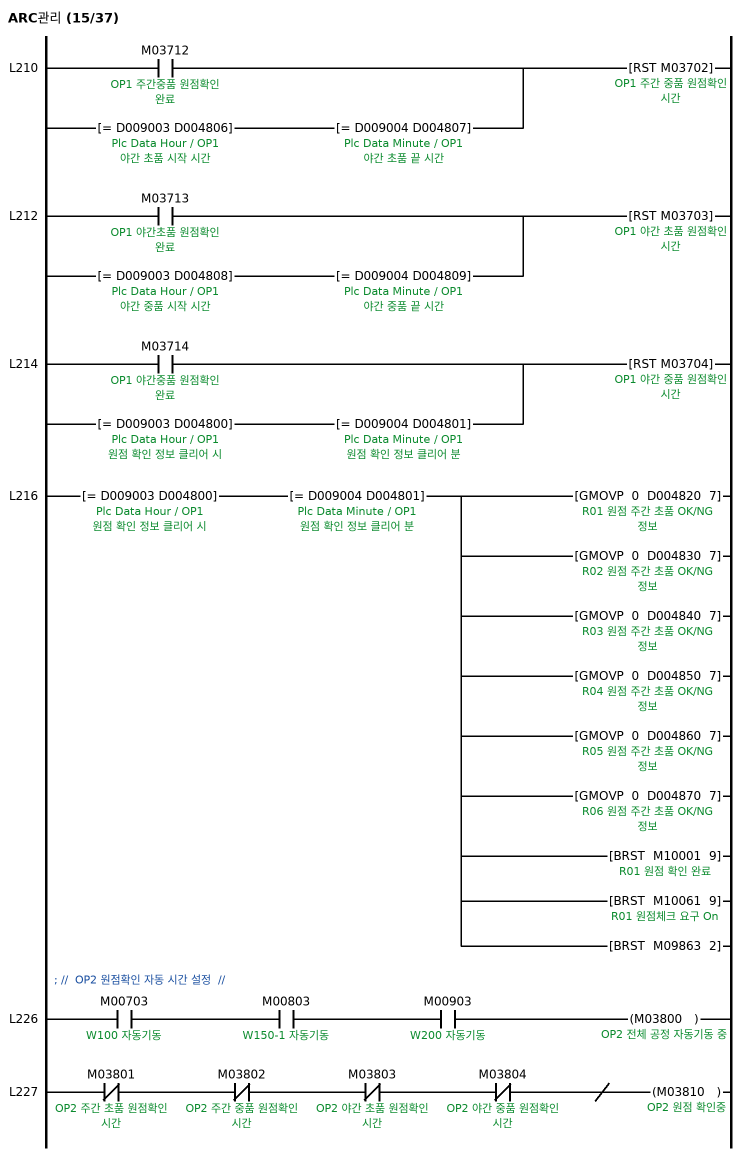
[picture p408: ARC관리 rungs L210-L227]
; L210
LOAD      M03712	// OP1 주간중품 원점확인 완료
LOAD=     D009003 D004806	// Plc Data Hour / OP1 야간 초품 시작 시간
AND=      D009004 D004807	// Plc Data Minute / OP1 야간 초품 끝 시간
OR LOAD
RST       M03702	// OP1 주간 중품 원점확인 시간
; L212
LOAD      M03713	// OP1 야간초품 원점확인 완료
LOAD=     D009003 D004808	// Plc Data Hour / OP1 야간 중품 시작 시간
AND=      D009004 D004809	// Plc Data Minute / OP1 야간 중품 끝 시간
OR LOAD
RST       M03703	// OP1 야간 초품 원점확인 시간
; L214
LOAD      M03714	// OP1 야간중품 원점확인 완료
LOAD=     D009003 D004800	// Plc Data Hour / OP1 원점 확인 정보 클리어 시
AND=      D009004 D004801	// Plc Data Minute / OP1 원점 확인 정보 클리어 분
OR LOAD
RST       M03704	// OP1 야간 중품 원점확인 시간
; L216
LOAD=     D009003 D004800	// Plc Data Hour / OP1 원점 확인 정보 클리어 시
AND=      D009004 D004801	// Plc Data Minute / OP1 원점 확인 정보 클리어 분
GMOVP     0 D004820 7	// R01 원점 주간 초품 OK/NG 정보
GMOVP     0 D004830 7	// R02 원점 주간 초품 OK/NG 정보
GMOVP     0 D004840 7	// R03 원점 주간 초품 OK/NG 정보
GMOVP     0 D004850 7	// R04 원점 주간 초품 OK/NG 정보
GMOVP     0 D004860 7	// R05 원점 주간 초품 OK/NG 정보
GMOVP     0 D004870 7	// R06 원점 주간 초품 OK/NG 정보
BRST      M10001 9	// R01 원점 확인 완료
BRST      M10061 9	// R01 원점체크 요구 On
BRST      M09863 2
//   //  OP2 원점확인 자동 시간 설정  //
; L226
LOAD      M00703	// W100 자동기동
AND       M00803	// W150-1 자동기동
AND       M00903	// W200 자동기동
OUT       M03800	// OP2 전체 공정 자동기동 중
; L227
LOAD NOT  M03801	// OP2 주간 초품 원점확인 시간
AND NOT   M03802	// OP2 주간 중품 원점확인 시간
AND NOT   M03803	// OP2 야간 초품 원점확인 시간
AND NOT   M03804	// OP2 야간 중품 원점확인 시간
NOT
OUT       M03810	// OP2 원점 확인중

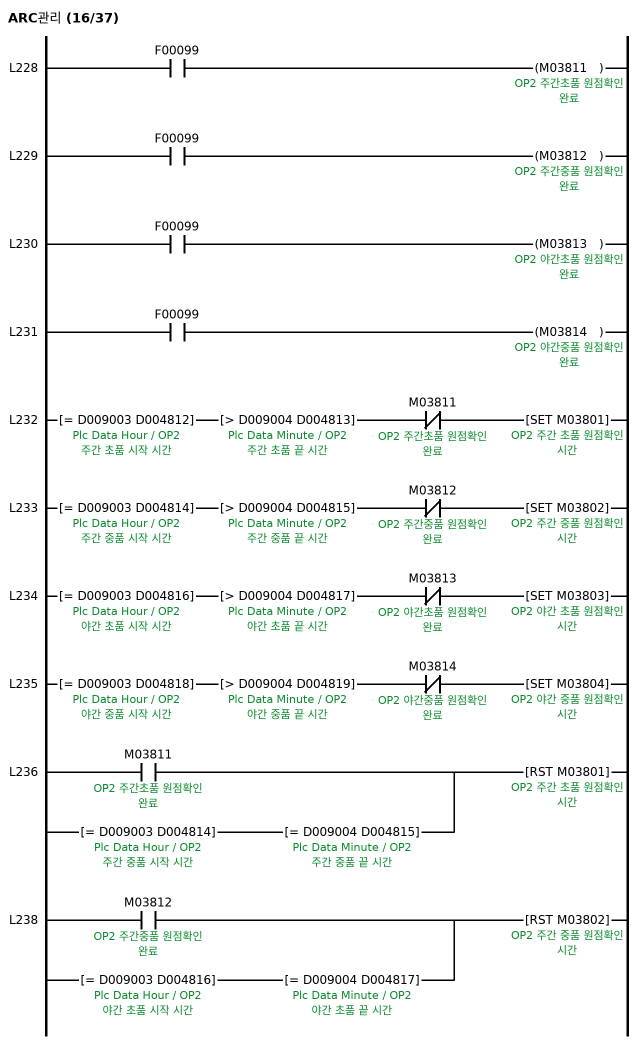
; L228
LOAD      F00099
OUT       M03811	// OP2 주간초품 원점확인 완료
; L229
LOAD      F00099
OUT       M03812	// OP2 주간중품 원점확인 완료
; L230
LOAD      F00099
OUT       M03813	// OP2 야간초품 원점확인 완료
; L231
LOAD      F00099
OUT       M03814	// OP2 야간중품 원점확인 완료
; L232
LOAD=     D009003 D004812	// Plc Data Hour / OP2 주간 초품 시작 시간
AND>      D009004 D004813	// Plc Data Minute / OP2 주간 초품 끝 시간
AND NOT   M03811	// OP2 주간초품 원점확인 완료
SET       M03801	// OP2 주간 초품 원점확인 시간
; L233
LOAD=     D009003 D004814	// Plc Data Hour / OP2 주간 중품 시작 시간
AND>      D009004 D004815	// Plc Data Minute / OP2 주간 중품 끝 시간
AND NOT   M03812	// OP2 주간중품 원점확인 완료
SET       M03802	// OP2 주간 중품 원점확인 시간
; L234
LOAD=     D009003 D004816	// Plc Data Hour / OP2 야간 초품 시작 시간
AND>      D009004 D004817	// Plc Data Minute / OP2 야간 초품 끝 시간
AND NOT   M03813	// OP2 야간초품 원점확인 완료
SET       M03803	// OP2 야간 초품 원점확인 시간
; L235
LOAD=     D009003 D004818	// Plc Data Hour / OP2 야간 중품 시작 시간
AND>      D009004 D004819	// Plc Data Minute / OP2 야간 중품 끝 시간
AND NOT   M03814	// OP2 야간중품 원점확인 완료
SET       M03804	// OP2 야간 중품 원점확인 시간
; L236
LOAD      M03811	// OP2 주간초품 원점확인 완료
LOAD=     D009003 D004814	// Plc Data Hour / OP2 주간 중품 시작 시간
AND=      D009004 D004815	// Plc Data Minute / OP2 주간 중품 끝 시간
OR LOAD
RST       M03801	// OP2 주간 초품 원점확인 시간
; L238
LOAD      M03812	// OP2 주간중품 원점확인 완료
LOAD=     D009003 D004816	// Plc Data Hour / OP2 야간 초품 시작 시간
AND=      D009004 D004817	// Plc Data Minute / OP2 야간 초품 끝 시간
OR LOAD
RST       M03802	// OP2 주간 중품 원점확인 시간

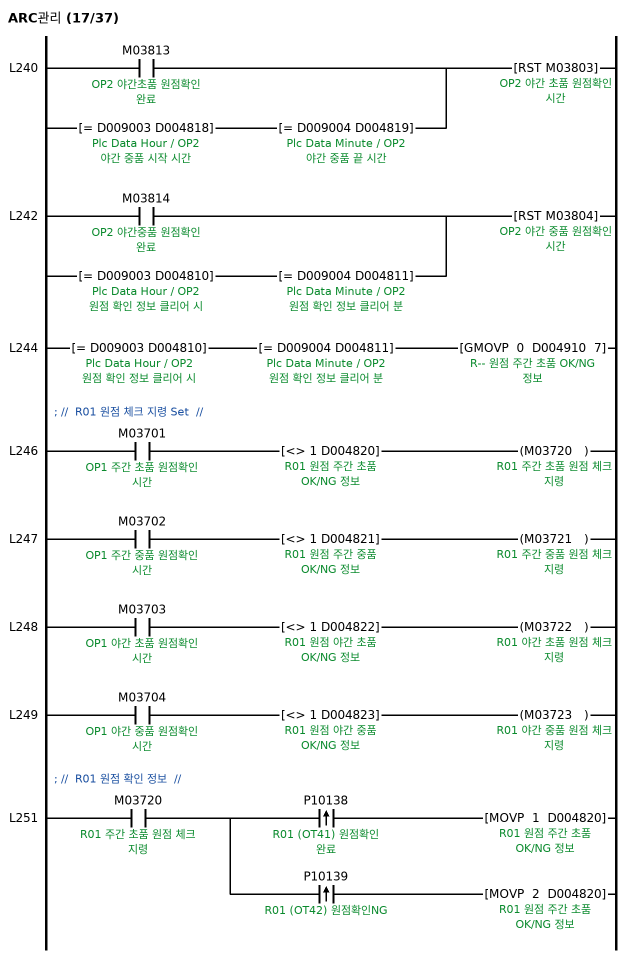
; L240
LOAD      M03813	// OP2 야간초품 원점확인 완료
LOAD=     D009003 D004818	// Plc Data Hour / OP2 야간 중품 시작 시간
AND=      D009004 D004819	// Plc Data Minute / OP2 야간 중품 끝 시간
OR LOAD
RST       M03803	// OP2 야간 초품 원점확인 시간
; L242
LOAD      M03814	// OP2 야간중품 원점확인 완료
LOAD=     D009003 D004810	// Plc Data Hour / OP2 원점 확인 정보 클리어 시
AND=      D009004 D004811	// Plc Data Minute / OP2 원점 확인 정보 클리어 분
OR LOAD
RST       M03804	// OP2 야간 중품 원점확인 시간
; L244
LOAD=     D009003 D004810	// Plc Data Hour / OP2 원점 확인 정보 클리어 시
AND=      D009004 D004811	// Plc Data Minute / OP2 원점 확인 정보 클리어 분
GMOVP     0 D004910 7	// R-- 원점 주간 초품 OK/NG 정보
//   //  R01 원점 체크 지령 Set  //
; L246
LOAD      M03701	// OP1 주간 초품 원점확인 시간
AND<>     1 D004820	// R01 원점 주간 초품 OK/NG 정보
OUT       M03720	// R01 주간 초품 원점 체크 지령
; L247
LOAD      M03702	// OP1 주간 중품 원점확인 시간
AND<>     1 D004821	// R01 원점 주간 중품 OK/NG 정보
OUT       M03721	// R01 주간 중품 원점 체크 지령
; L248
LOAD      M03703	// OP1 야간 초품 원점확인 시간
AND<>     1 D004822	// R01 원점 야간 초품 OK/NG 정보
OUT       M03722	// R01 야간 초품 원점 체크 지령
; L249
LOAD      M03704	// OP1 야간 중품 원점확인 시간
AND<>     1 D004823	// R01 원점 야간 중품 OK/NG 정보
OUT       M03723	// R01 야간 중품 원점 체크 지령
//   //  R01 원점 확인 정보  //
; L251
LOAD      M03720	// R01 주간 초품 원점 체크 지령
MPUSH
ANDP      P10138	// R01 (OT41) 원점확인 완료
MOVP      1 D004820	// R01 원점 주간 초품 OK/NG 정보
MPOP
ANDP      P10139	// R01 (OT42) 원점확인NG
MOVP      2 D004820	// R01 원점 주간 초품 OK/NG 정보

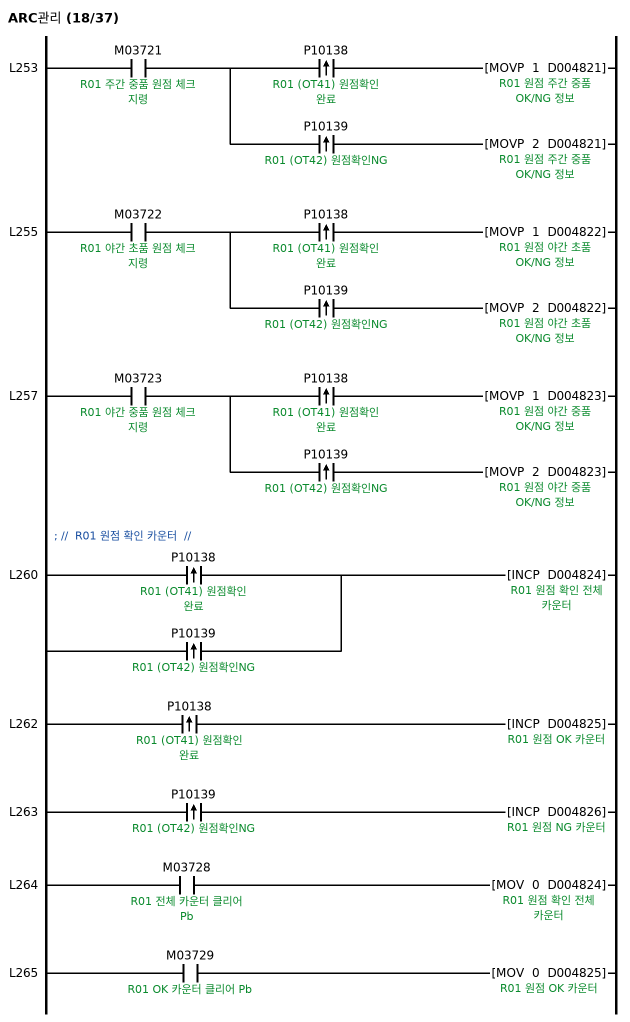
; L253
LOAD      M03721	// R01 주간 중품 원점 체크 지령
MPUSH
ANDP      P10138	// R01 (OT41) 원점확인 완료
MOVP      1 D004821	// R01 원점 주간 중품 OK/NG 정보
MPOP
ANDP      P10139	// R01 (OT42) 원점확인NG
MOVP      2 D004821	// R01 원점 주간 중품 OK/NG 정보
; L255
LOAD      M03722	// R01 야간 초품 원점 체크 지령
MPUSH
ANDP      P10138	// R01 (OT41) 원점확인 완료
MOVP      1 D004822	// R01 원점 야간 초품 OK/NG 정보
MPOP
ANDP      P10139	// R01 (OT42) 원점확인NG
MOVP      2 D004822	// R01 원점 야간 초품 OK/NG 정보
; L257
LOAD      M03723	// R01 야간 중품 원점 체크 지령
MPUSH
ANDP      P10138	// R01 (OT41) 원점확인 완료
MOVP      1 D004823	// R01 원점 야간 중품 OK/NG 정보
MPOP
ANDP      P10139	// R01 (OT42) 원점확인NG
MOVP      2 D004823	// R01 원점 야간 중품 OK/NG 정보
//   //  R01 원점 확인 카운터  //
; L260
LOADP     P10138	// R01 (OT41) 원점확인 완료
ORP       P10139	// R01 (OT42) 원점확인NG
INCP      D004824	// R01 원점 확인 전체 카운터
; L262
LOADP     P10138	// R01 (OT41) 원점확인 완료
INCP      D004825	// R01 원점 OK 카운터
; L263
LOADP     P10139	// R01 (OT42) 원점확인NG
INCP      D004826	// R01 원점 NG 카운터
; L264
LOAD      M03728	// R01 전체 카운터 클리어 Pb
MOV       0 D004824	// R01 원점 확인 전체 카운터
; L265
LOAD      M03729	// R01 OK 카운터 클리어 Pb
MOV       0 D004825	// R01 원점 OK 카운터

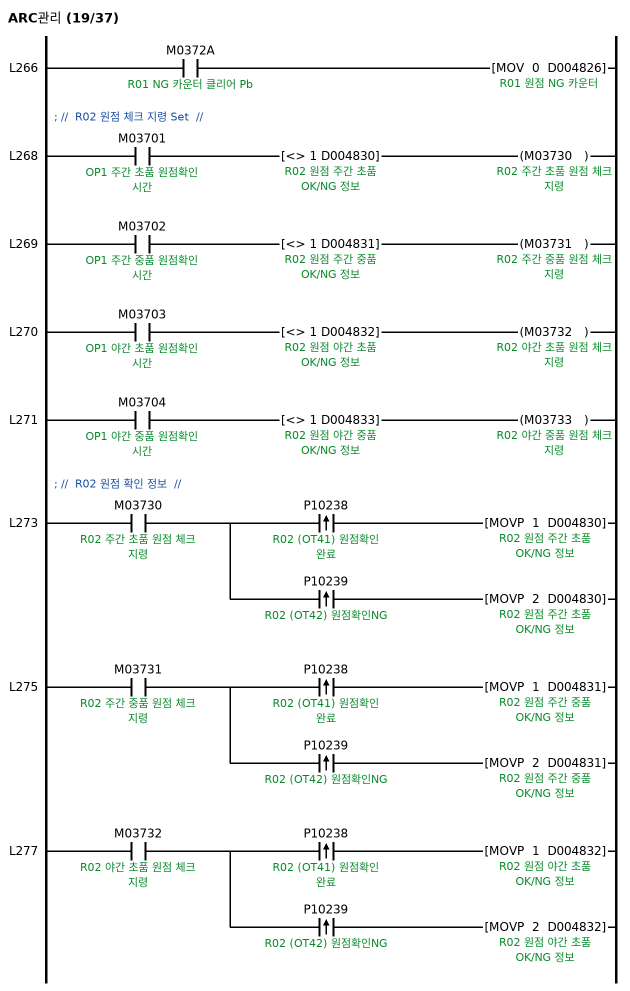
; L266
LOAD      M0372A	// R01 NG 카운터 클리어 Pb
MOV       0 D004826	// R01 원점 NG 카운터
//   //  R02 원점 체크 지령 Set  //
; L268
LOAD      M03701	// OP1 주간 초품 원점확인 시간
AND<>     1 D004830	// R02 원점 주간 초품 OK/NG 정보
OUT       M03730	// R02 주간 초품 원점 체크 지령
; L269
LOAD      M03702	// OP1 주간 중품 원점확인 시간
AND<>     1 D004831	// R02 원점 주간 중품 OK/NG 정보
OUT       M03731	// R02 주간 중품 원점 체크 지령
; L270
LOAD      M03703	// OP1 야간 초품 원점확인 시간
AND<>     1 D004832	// R02 원점 야간 초품 OK/NG 정보
OUT       M03732	// R02 야간 초품 원점 체크 지령
; L271
LOAD      M03704	// OP1 야간 중품 원점확인 시간
AND<>     1 D004833	// R02 원점 야간 중품 OK/NG 정보
OUT       M03733	// R02 야간 중품 원점 체크 지령
//   //  R02 원점 확인 정보  //
; L273
LOAD      M03730	// R02 주간 초품 원점 체크 지령
MPUSH
ANDP      P10238	// R02 (OT41) 원점확인 완료
MOVP      1 D004830	// R02 원점 주간 초품 OK/NG 정보
MPOP
ANDP      P10239	// R02 (OT42) 원점확인NG
MOVP      2 D004830	// R02 원점 주간 초품 OK/NG 정보
; L275
LOAD      M03731	// R02 주간 중품 원점 체크 지령
MPUSH
ANDP      P10238	// R02 (OT41) 원점확인 완료
MOVP      1 D004831	// R02 원점 주간 중품 OK/NG 정보
MPOP
ANDP      P10239	// R02 (OT42) 원점확인NG
MOVP      2 D004831	// R02 원점 주간 중품 OK/NG 정보
; L277
LOAD      M03732	// R02 야간 초품 원점 체크 지령
MPUSH
ANDP      P10238	// R02 (OT41) 원점확인 완료
MOVP      1 D004832	// R02 원점 야간 초품 OK/NG 정보
MPOP
ANDP      P10239	// R02 (OT42) 원점확인NG
MOVP      2 D004832	// R02 원점 야간 초품 OK/NG 정보

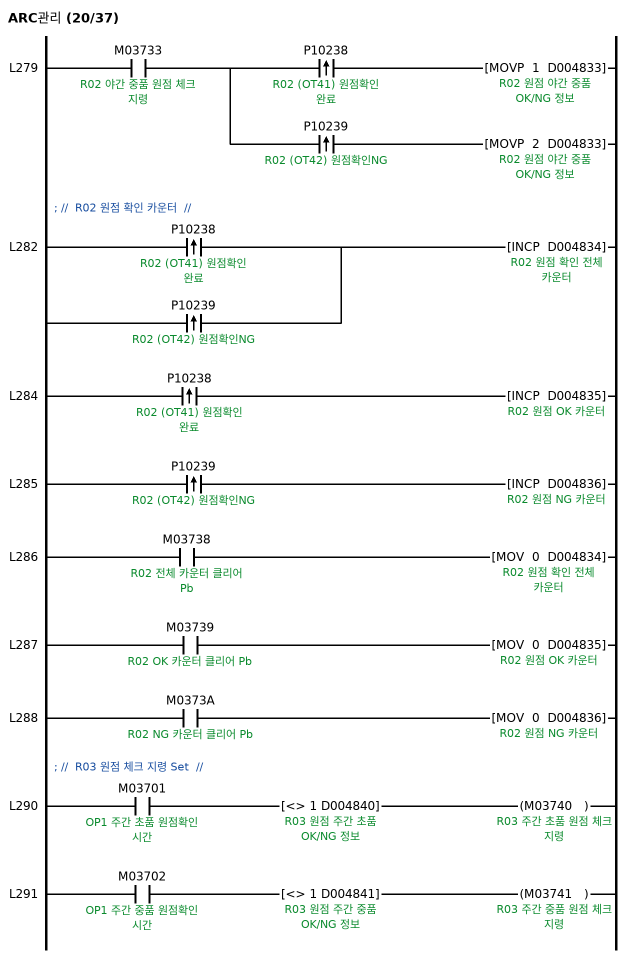
; L279
LOAD      M03733	// R02 야간 중품 원점 체크 지령
MPUSH
ANDP      P10238	// R02 (OT41) 원점확인 완료
MOVP      1 D004833	// R02 원점 야간 중품 OK/NG 정보
MPOP
ANDP      P10239	// R02 (OT42) 원점확인NG
MOVP      2 D004833	// R02 원점 야간 중품 OK/NG 정보
//   //  R02 원점 확인 카운터  //
; L282
LOADP     P10238	// R02 (OT41) 원점확인 완료
ORP       P10239	// R02 (OT42) 원점확인NG
INCP      D004834	// R02 원점 확인 전체 카운터
; L284
LOADP     P10238	// R02 (OT41) 원점확인 완료
INCP      D004835	// R02 원점 OK 카운터
; L285
LOADP     P10239	// R02 (OT42) 원점확인NG
INCP      D004836	// R02 원점 NG 카운터
; L286
LOAD      M03738	// R02 전체 카운터 클리어 Pb
MOV       0 D004834	// R02 원점 확인 전체 카운터
; L287
LOAD      M03739	// R02 OK 카운터 클리어 Pb
MOV       0 D004835	// R02 원점 OK 카운터
; L288
LOAD      M0373A	// R02 NG 카운터 클리어 Pb
MOV       0 D004836	// R02 원점 NG 카운터
//   //  R03 원점 체크 지령 Set  //
; L290
LOAD      M03701	// OP1 주간 초품 원점확인 시간
AND<>     1 D004840	// R03 원점 주간 초품 OK/NG 정보
OUT       M03740	// R03 주간 초품 원점 체크 지령
; L291
LOAD      M03702	// OP1 주간 중품 원점확인 시간
AND<>     1 D004841	// R03 원점 주간 중품 OK/NG 정보
OUT       M03741	// R03 주간 중품 원점 체크 지령

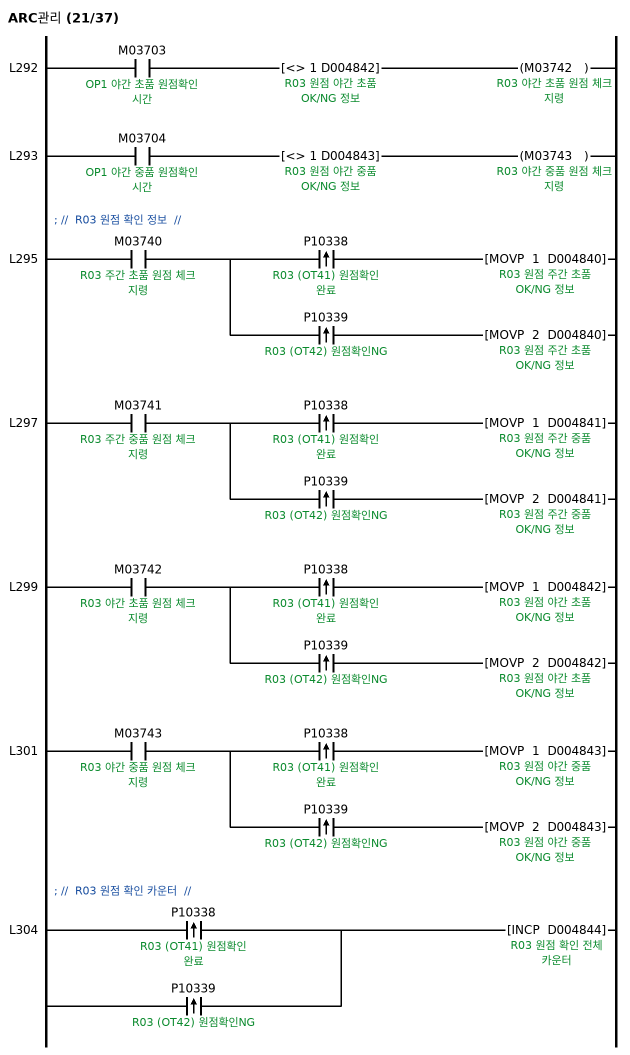
; L292
LOAD      M03703	// OP1 야간 초품 원점확인 시간
AND<>     1 D004842	// R03 원점 야간 초품 OK/NG 정보
OUT       M03742	// R03 야간 초품 원점 체크 지령
; L293
LOAD      M03704	// OP1 야간 중품 원점확인 시간
AND<>     1 D004843	// R03 원점 야간 중품 OK/NG 정보
OUT       M03743	// R03 야간 중품 원점 체크 지령
//   //  R03 원점 확인 정보  //
; L295
LOAD      M03740	// R03 주간 초품 원점 체크 지령
MPUSH
ANDP      P10338	// R03 (OT41) 원점확인 완료
MOVP      1 D004840	// R03 원점 주간 초품 OK/NG 정보
MPOP
ANDP      P10339	// R03 (OT42) 원점확인NG
MOVP      2 D004840	// R03 원점 주간 초품 OK/NG 정보
; L297
LOAD      M03741	// R03 주간 중품 원점 체크 지령
MPUSH
ANDP      P10338	// R03 (OT41) 원점확인 완료
MOVP      1 D004841	// R03 원점 주간 중품 OK/NG 정보
MPOP
ANDP      P10339	// R03 (OT42) 원점확인NG
MOVP      2 D004841	// R03 원점 주간 중품 OK/NG 정보
; L299
LOAD      M03742	// R03 야간 초품 원점 체크 지령
MPUSH
ANDP      P10338	// R03 (OT41) 원점확인 완료
MOVP      1 D004842	// R03 원점 야간 초품 OK/NG 정보
MPOP
ANDP      P10339	// R03 (OT42) 원점확인NG
MOVP      2 D004842	// R03 원점 야간 초품 OK/NG 정보
; L301
LOAD      M03743	// R03 야간 중품 원점 체크 지령
MPUSH
ANDP      P10338	// R03 (OT41) 원점확인 완료
MOVP      1 D004843	// R03 원점 야간 중품 OK/NG 정보
MPOP
ANDP      P10339	// R03 (OT42) 원점확인NG
MOVP      2 D004843	// R03 원점 야간 중품 OK/NG 정보
//   //  R03 원점 확인 카운터  //
; L304
LOADP     P10338	// R03 (OT41) 원점확인 완료
ORP       P10339	// R03 (OT42) 원점확인NG
INCP      D004844	// R03 원점 확인 전체 카운터

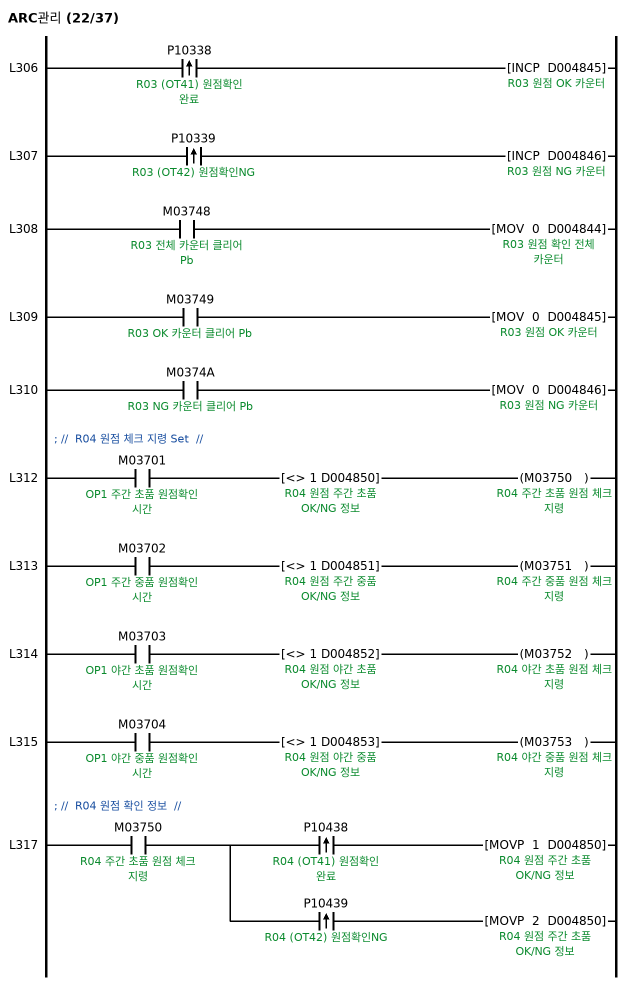
; L306
LOADP     P10338	// R03 (OT41) 원점확인 완료
INCP      D004845	// R03 원점 OK 카운터
; L307
LOADP     P10339	// R03 (OT42) 원점확인NG
INCP      D004846	// R03 원점 NG 카운터
; L308
LOAD      M03748	// R03 전체 카운터 클리어 Pb
MOV       0 D004844	// R03 원점 확인 전체 카운터
; L309
LOAD      M03749	// R03 OK 카운터 클리어 Pb
MOV       0 D004845	// R03 원점 OK 카운터
; L310
LOAD      M0374A	// R03 NG 카운터 클리어 Pb
MOV       0 D004846	// R03 원점 NG 카운터
//   //  R04 원점 체크 지령 Set  //
; L312
LOAD      M03701	// OP1 주간 초품 원점확인 시간
AND<>     1 D004850	// R04 원점 주간 초품 OK/NG 정보
OUT       M03750	// R04 주간 초품 원점 체크 지령
; L313
LOAD      M03702	// OP1 주간 중품 원점확인 시간
AND<>     1 D004851	// R04 원점 주간 중품 OK/NG 정보
OUT       M03751	// R04 주간 중품 원점 체크 지령
; L314
LOAD      M03703	// OP1 야간 초품 원점확인 시간
AND<>     1 D004852	// R04 원점 야간 초품 OK/NG 정보
OUT       M03752	// R04 야간 초품 원점 체크 지령
; L315
LOAD      M03704	// OP1 야간 중품 원점확인 시간
AND<>     1 D004853	// R04 원점 야간 중품 OK/NG 정보
OUT       M03753	// R04 야간 중품 원점 체크 지령
//   //  R04 원점 확인 정보  //
; L317
LOAD      M03750	// R04 주간 초품 원점 체크 지령
MPUSH
ANDP      P10438	// R04 (OT41) 원점확인 완료
MOVP      1 D004850	// R04 원점 주간 초품 OK/NG 정보
MPOP
ANDP      P10439	// R04 (OT42) 원점확인NG
MOVP      2 D004850	// R04 원점 주간 초품 OK/NG 정보

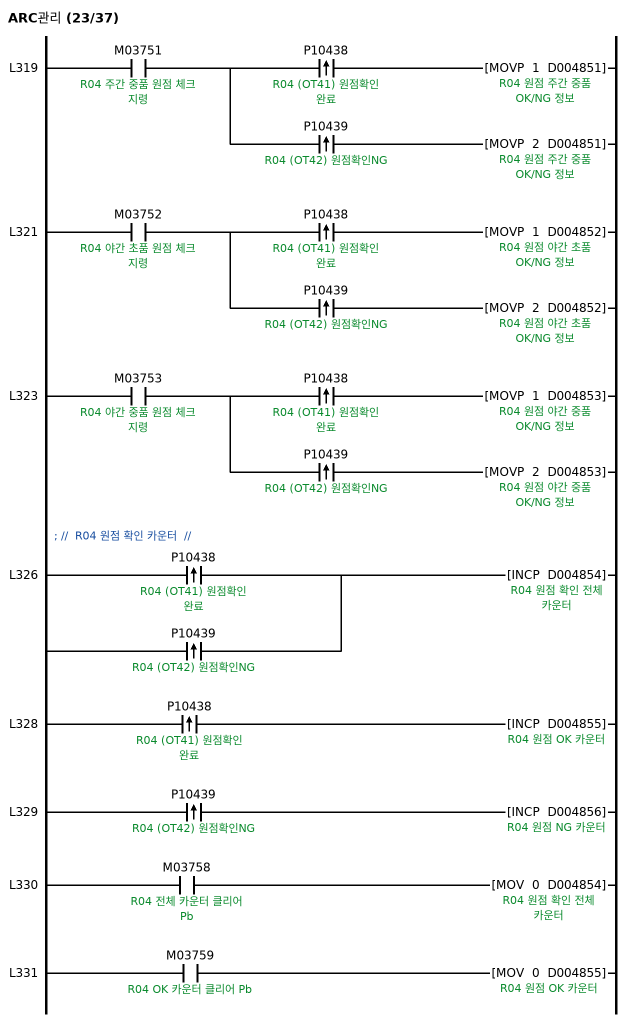
; L319
LOAD      M03751	// R04 주간 중품 원점 체크 지령
MPUSH
ANDP      P10438	// R04 (OT41) 원점확인 완료
MOVP      1 D004851	// R04 원점 주간 중품 OK/NG 정보
MPOP
ANDP      P10439	// R04 (OT42) 원점확인NG
MOVP      2 D004851	// R04 원점 주간 중품 OK/NG 정보
; L321
LOAD      M03752	// R04 야간 초품 원점 체크 지령
MPUSH
ANDP      P10438	// R04 (OT41) 원점확인 완료
MOVP      1 D004852	// R04 원점 야간 초품 OK/NG 정보
MPOP
ANDP      P10439	// R04 (OT42) 원점확인NG
MOVP      2 D004852	// R04 원점 야간 초품 OK/NG 정보
; L323
LOAD      M03753	// R04 야간 중품 원점 체크 지령
MPUSH
ANDP      P10438	// R04 (OT41) 원점확인 완료
MOVP      1 D004853	// R04 원점 야간 중품 OK/NG 정보
MPOP
ANDP      P10439	// R04 (OT42) 원점확인NG
MOVP      2 D004853	// R04 원점 야간 중품 OK/NG 정보
//   //  R04 원점 확인 카운터  //
; L326
LOADP     P10438	// R04 (OT41) 원점확인 완료
ORP       P10439	// R04 (OT42) 원점확인NG
INCP      D004854	// R04 원점 확인 전체 카운터
; L328
LOADP     P10438	// R04 (OT41) 원점확인 완료
INCP      D004855	// R04 원점 OK 카운터
; L329
LOADP     P10439	// R04 (OT42) 원점확인NG
INCP      D004856	// R04 원점 NG 카운터
; L330
LOAD      M03758	// R04 전체 카운터 클리어 Pb
MOV       0 D004854	// R04 원점 확인 전체 카운터
; L331
LOAD      M03759	// R04 OK 카운터 클리어 Pb
MOV       0 D004855	// R04 원점 OK 카운터

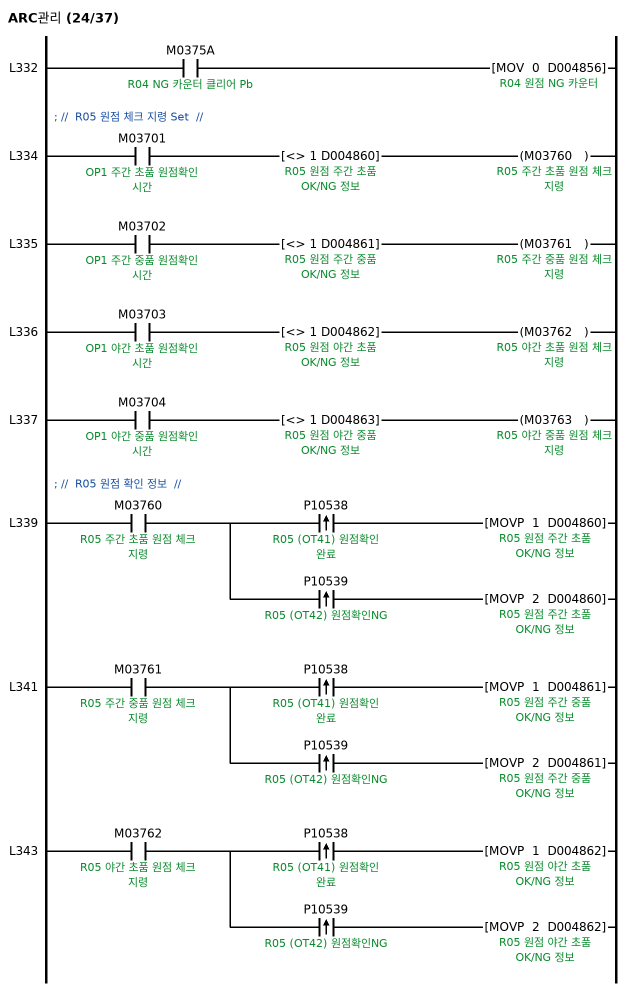
; L332
LOAD      M0375A	// R04 NG 카운터 클리어 Pb
MOV       0 D004856	// R04 원점 NG 카운터
//   //  R05 원점 체크 지령 Set  //
; L334
LOAD      M03701	// OP1 주간 초품 원점확인 시간
AND<>     1 D004860	// R05 원점 주간 초품 OK/NG 정보
OUT       M03760	// R05 주간 초품 원점 체크 지령
; L335
LOAD      M03702	// OP1 주간 중품 원점확인 시간
AND<>     1 D004861	// R05 원점 주간 중품 OK/NG 정보
OUT       M03761	// R05 주간 중품 원점 체크 지령
; L336
LOAD      M03703	// OP1 야간 초품 원점확인 시간
AND<>     1 D004862	// R05 원점 야간 초품 OK/NG 정보
OUT       M03762	// R05 야간 초품 원점 체크 지령
; L337
LOAD      M03704	// OP1 야간 중품 원점확인 시간
AND<>     1 D004863	// R05 원점 야간 중품 OK/NG 정보
OUT       M03763	// R05 야간 중품 원점 체크 지령
//   //  R05 원점 확인 정보  //
; L339
LOAD      M03760	// R05 주간 초품 원점 체크 지령
MPUSH
ANDP      P10538	// R05 (OT41) 원점확인 완료
MOVP      1 D004860	// R05 원점 주간 초품 OK/NG 정보
MPOP
ANDP      P10539	// R05 (OT42) 원점확인NG
MOVP      2 D004860	// R05 원점 주간 초품 OK/NG 정보
; L341
LOAD      M03761	// R05 주간 중품 원점 체크 지령
MPUSH
ANDP      P10538	// R05 (OT41) 원점확인 완료
MOVP      1 D004861	// R05 원점 주간 중품 OK/NG 정보
MPOP
ANDP      P10539	// R05 (OT42) 원점확인NG
MOVP      2 D004861	// R05 원점 주간 중품 OK/NG 정보
; L343
LOAD      M03762	// R05 야간 초품 원점 체크 지령
MPUSH
ANDP      P10538	// R05 (OT41) 원점확인 완료
MOVP      1 D004862	// R05 원점 야간 초품 OK/NG 정보
MPOP
ANDP      P10539	// R05 (OT42) 원점확인NG
MOVP      2 D004862	// R05 원점 야간 초품 OK/NG 정보

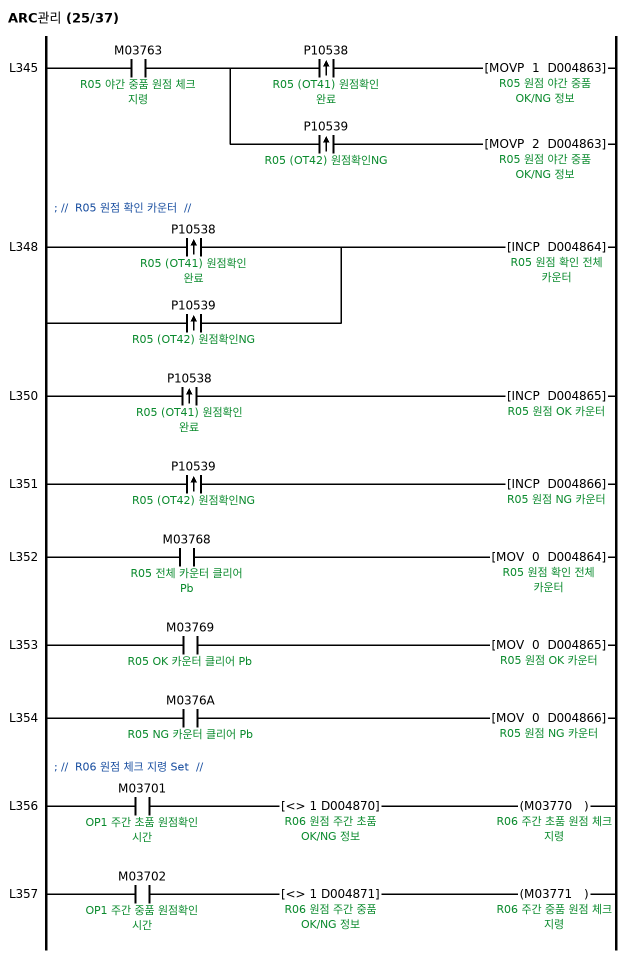
; L345
LOAD      M03763	// R05 야간 중품 원점 체크 지령
MPUSH
ANDP      P10538	// R05 (OT41) 원점확인 완료
MOVP      1 D004863	// R05 원점 야간 중품 OK/NG 정보
MPOP
ANDP      P10539	// R05 (OT42) 원점확인NG
MOVP      2 D004863	// R05 원점 야간 중품 OK/NG 정보
//   //  R05 원점 확인 카운터  //
; L348
LOADP     P10538	// R05 (OT41) 원점확인 완료
ORP       P10539	// R05 (OT42) 원점확인NG
INCP      D004864	// R05 원점 확인 전체 카운터
; L350
LOADP     P10538	// R05 (OT41) 원점확인 완료
INCP      D004865	// R05 원점 OK 카운터
; L351
LOADP     P10539	// R05 (OT42) 원점확인NG
INCP      D004866	// R05 원점 NG 카운터
; L352
LOAD      M03768	// R05 전체 카운터 클리어 Pb
MOV       0 D004864	// R05 원점 확인 전체 카운터
; L353
LOAD      M03769	// R05 OK 카운터 클리어 Pb
MOV       0 D004865	// R05 원점 OK 카운터
; L354
LOAD      M0376A	// R05 NG 카운터 클리어 Pb
MOV       0 D004866	// R05 원점 NG 카운터
//   //  R06 원점 체크 지령 Set  //
; L356
LOAD      M03701	// OP1 주간 초품 원점확인 시간
AND<>     1 D004870	// R06 원점 주간 초품 OK/NG 정보
OUT       M03770	// R06 주간 초품 원점 체크 지령
; L357
LOAD      M03702	// OP1 주간 중품 원점확인 시간
AND<>     1 D004871	// R06 원점 주간 중품 OK/NG 정보
OUT       M03771	// R06 주간 중품 원점 체크 지령

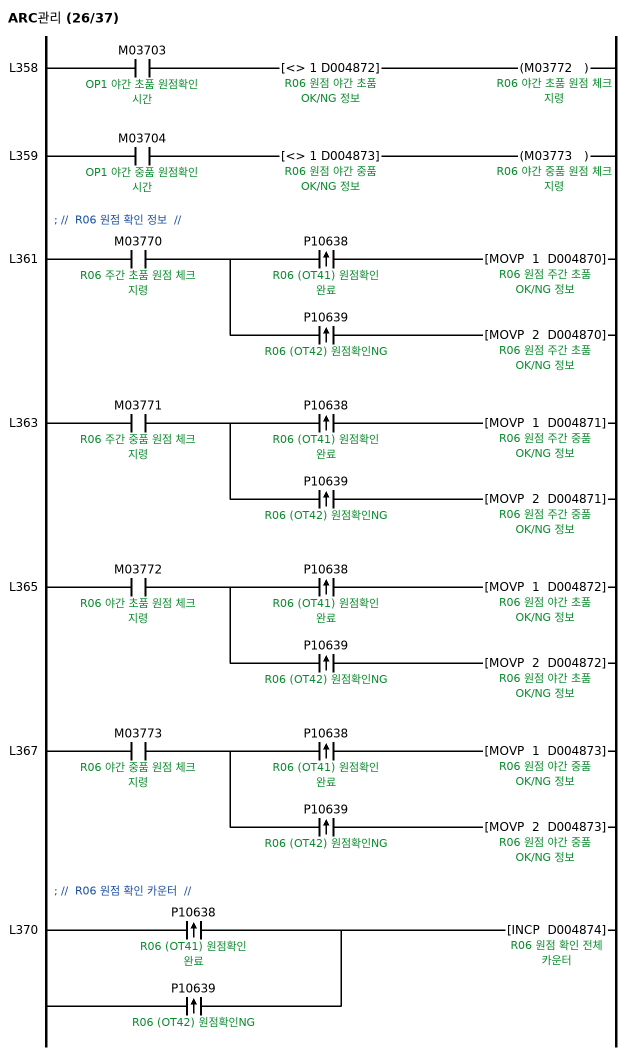
; L358
LOAD      M03703	// OP1 야간 초품 원점확인 시간
AND<>     1 D004872	// R06 원점 야간 초품 OK/NG 정보
OUT       M03772	// R06 야간 초품 원점 체크 지령
; L359
LOAD      M03704	// OP1 야간 중품 원점확인 시간
AND<>     1 D004873	// R06 원점 야간 중품 OK/NG 정보
OUT       M03773	// R06 야간 중품 원점 체크 지령
//   //  R06 원점 확인 정보  //
; L361
LOAD      M03770	// R06 주간 초품 원점 체크 지령
MPUSH
ANDP      P10638	// R06 (OT41) 원점확인 완료
MOVP      1 D004870	// R06 원점 주간 초품 OK/NG 정보
MPOP
ANDP      P10639	// R06 (OT42) 원점확인NG
MOVP      2 D004870	// R06 원점 주간 초품 OK/NG 정보
; L363
LOAD      M03771	// R06 주간 중품 원점 체크 지령
MPUSH
ANDP      P10638	// R06 (OT41) 원점확인 완료
MOVP      1 D004871	// R06 원점 주간 중품 OK/NG 정보
MPOP
ANDP      P10639	// R06 (OT42) 원점확인NG
MOVP      2 D004871	// R06 원점 주간 중품 OK/NG 정보
; L365
LOAD      M03772	// R06 야간 초품 원점 체크 지령
MPUSH
ANDP      P10638	// R06 (OT41) 원점확인 완료
MOVP      1 D004872	// R06 원점 야간 초품 OK/NG 정보
MPOP
ANDP      P10639	// R06 (OT42) 원점확인NG
MOVP      2 D004872	// R06 원점 야간 초품 OK/NG 정보
; L367
LOAD      M03773	// R06 야간 중품 원점 체크 지령
MPUSH
ANDP      P10638	// R06 (OT41) 원점확인 완료
MOVP      1 D004873	// R06 원점 야간 중품 OK/NG 정보
MPOP
ANDP      P10639	// R06 (OT42) 원점확인NG
MOVP      2 D004873	// R06 원점 야간 중품 OK/NG 정보
//   //  R06 원점 확인 카운터  //
; L370
LOADP     P10638	// R06 (OT41) 원점확인 완료
ORP       P10639	// R06 (OT42) 원점확인NG
INCP      D004874	// R06 원점 확인 전체 카운터

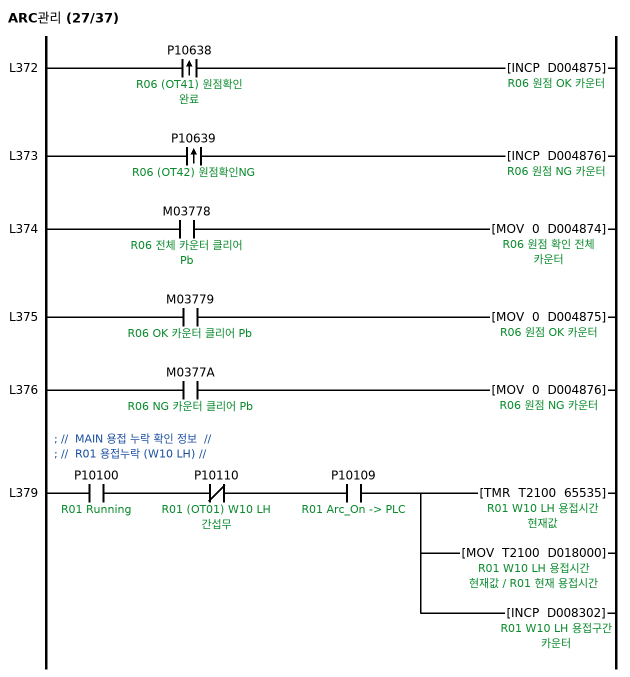
; L372
LOADP     P10638	// R06 (OT41) 원점확인 완료
INCP      D004875	// R06 원점 OK 카운터
; L373
LOADP     P10639	// R06 (OT42) 원점확인NG
INCP      D004876	// R06 원점 NG 카운터
; L374
LOAD      M03778	// R06 전체 카운터 클리어 Pb
MOV       0 D004874	// R06 원점 확인 전체 카운터
; L375
LOAD      M03779	// R06 OK 카운터 클리어 Pb
MOV       0 D004875	// R06 원점 OK 카운터
; L376
LOAD      M0377A	// R06 NG 카운터 클리어 Pb
MOV       0 D004876	// R06 원점 NG 카운터
//   //  MAIN 용접 누락 확인 정보  //
//   //  R01 용접누락 (W10 LH) //
; L379
LOAD      P10100	// R01 Running
AND NOT   P10110	// R01 (OT01) W10 LH 간섭무
AND       P10109	// R01 Arc_On -> PLC
TMR       T2100 65535	// R01 W10 LH 용접시간 현재값
MOV       T2100 D018000	// R01 W10 LH 용접시간 현재값 / R01 현재 용접시간
INCP      D008302	// R01 W10 LH 용접구간 카운터

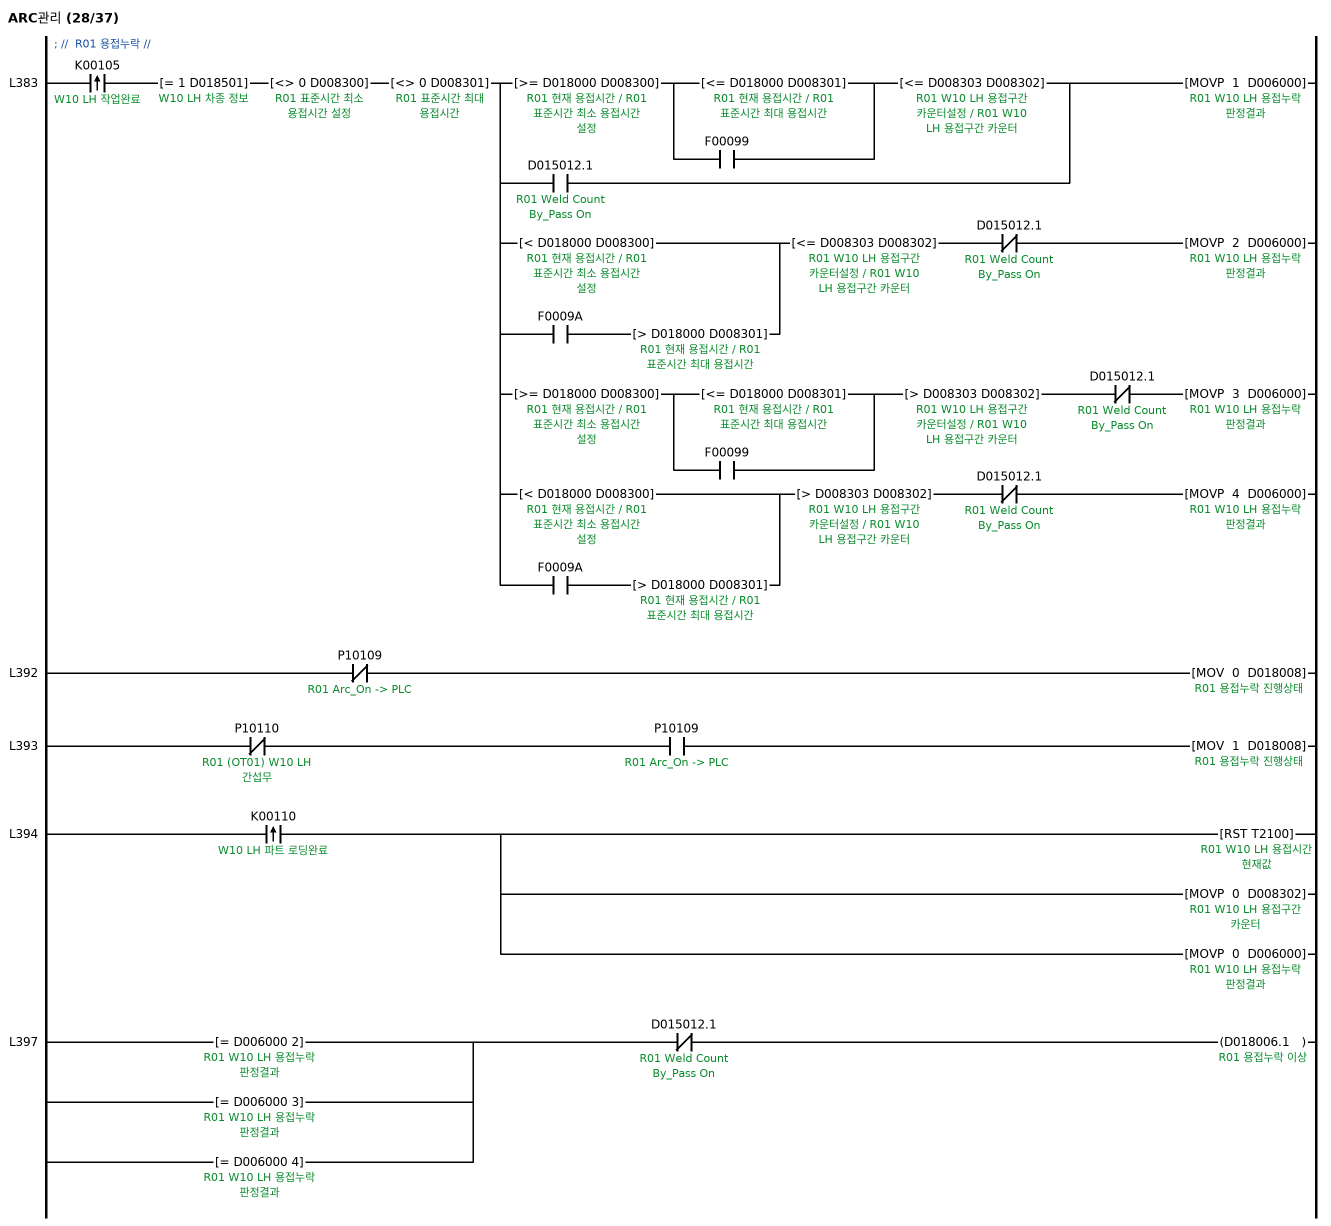
//   //  R01 용접누락 //
; L383
LOADP     K00105	// W10 LH 작업완료
AND=      1 D018501	// W10 LH 차종 정보
AND<>     0 D008300	// R01 표준시간 최소 용접시간 설정
AND<>     0 D008301	// R01 표준시간 최대 용접시간
MPUSH
LOAD>=    D018000 D008300	// R01 현재 용접시간 / R01 표준시간 최소 용접시간 설정
LOAD<=    D018000 D008301	// R01 현재 용접시간 / R01 표준시간 최대 용접시간
OR        F00099
AND LOAD
AND<=     D008303 D008302	// R01 W10 LH 용접구간 카운터설정 / R01 W10 LH 용접구간 카운터
OR        D015012.1	// R01 Weld Count By_Pass On
AND LOAD
MOVP      1 D006000	// R01 W10 LH 용접누락 판정결과
MLOAD
LOAD<     D018000 D008300	// R01 현재 용접시간 / R01 표준시간 최소 용접시간 설정
LOAD      F0009A
AND>      D018000 D008301	// R01 현재 용접시간 / R01 표준시간 최대 용접시간
OR LOAD
AND LOAD
AND<=     D008303 D008302	// R01 W10 LH 용접구간 카운터설정 / R01 W10 LH 용접구간 카운터
AND NOT   D015012.1	// R01 Weld Count By_Pass On
MOVP      2 D006000	// R01 W10 LH 용접누락 판정결과
MLOAD
AND>=     D018000 D008300	// R01 현재 용접시간 / R01 표준시간 최소 용접시간 설정
LOAD<=    D018000 D008301	// R01 현재 용접시간 / R01 표준시간 최대 용접시간
OR        F00099
AND LOAD
AND>      D008303 D008302	// R01 W10 LH 용접구간 카운터설정 / R01 W10 LH 용접구간 카운터
AND NOT   D015012.1	// R01 Weld Count By_Pass On
MOVP      3 D006000	// R01 W10 LH 용접누락 판정결과
MPOP
LOAD<     D018000 D008300	// R01 현재 용접시간 / R01 표준시간 최소 용접시간 설정
LOAD      F0009A
AND>      D018000 D008301	// R01 현재 용접시간 / R01 표준시간 최대 용접시간
OR LOAD
AND LOAD
AND>      D008303 D008302	// R01 W10 LH 용접구간 카운터설정 / R01 W10 LH 용접구간 카운터
AND NOT   D015012.1	// R01 Weld Count By_Pass On
MOVP      4 D006000	// R01 W10 LH 용접누락 판정결과
; L392
LOAD NOT  P10109	// R01 Arc_On -> PLC
MOV       0 D018008	// R01 용접누락 진행상태
; L393
LOAD NOT  P10110	// R01 (OT01) W10 LH 간섭무
AND       P10109	// R01 Arc_On -> PLC
MOV       1 D018008	// R01 용접누락 진행상태
; L394
LOADP     K00110	// W10 LH 파트 로딩완료
RST       T2100	// R01 W10 LH 용접시간 현재값
MOVP      0 D008302	// R01 W10 LH 용접구간 카운터
MOVP      0 D006000	// R01 W10 LH 용접누락 판정결과
; L397
LOAD=     D006000 2	// R01 W10 LH 용접누락 판정결과
OR=       D006000 3	// R01 W10 LH 용접누락 판정결과
OR=       D006000 4	// R01 W10 LH 용접누락 판정결과
AND NOT   D015012.1	// R01 Weld Count By_Pass On
OUT       D018006.1	// R01 용접누락 이상

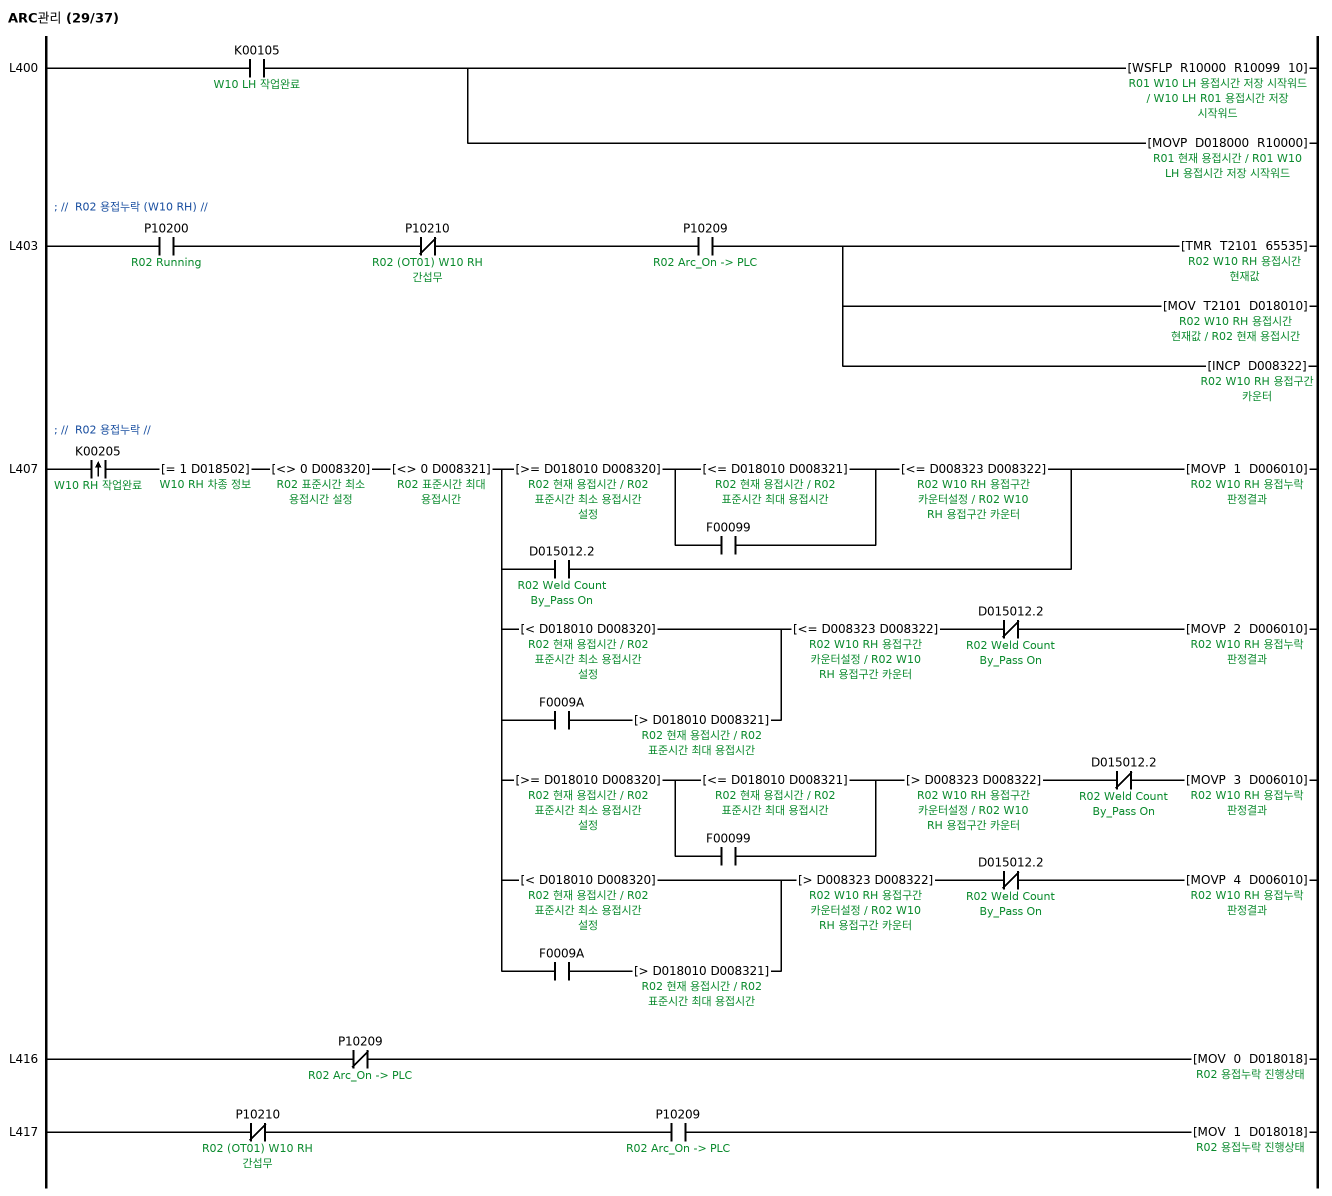
; L400
LOAD      K00105	// W10 LH 작업완료
WSFLP     R10000 R10099 10	// R01 W10 LH 용접시간 저장 시작워드 / W10 LH R01 용접시간 저장 시작워드
MOVP      D018000 R10000	// R01 현재 용접시간 / R01 W10 LH 용접시간 저장 시작워드
//   //  R02 용접누락 (W10 RH) //
; L403
LOAD      P10200	// R02 Running
AND NOT   P10210	// R02 (OT01) W10 RH 간섭무
AND       P10209	// R02 Arc_On -> PLC
TMR       T2101 65535	// R02 W10 RH 용접시간 현재값
MOV       T2101 D018010	// R02 W10 RH 용접시간 현재값 / R02 현재 용접시간
INCP      D008322	// R02 W10 RH 용접구간 카운터
//   //  R02 용접누락 //
; L407
LOADP     K00205	// W10 RH 작업완료
AND=      1 D018502	// W10 RH 차종 정보
AND<>     0 D008320	// R02 표준시간 최소 용접시간 설정
AND<>     0 D008321	// R02 표준시간 최대 용접시간
MPUSH
LOAD>=    D018010 D008320	// R02 현재 용접시간 / R02 표준시간 최소 용접시간 설정
LOAD<=    D018010 D008321	// R02 현재 용접시간 / R02 표준시간 최대 용접시간
OR        F00099
AND LOAD
AND<=     D008323 D008322	// R02 W10 RH 용접구간 카운터설정 / R02 W10 RH 용접구간 카운터
OR        D015012.2	// R02 Weld Count By_Pass On
AND LOAD
MOVP      1 D006010	// R02 W10 RH 용접누락 판정결과
MLOAD
LOAD<     D018010 D008320	// R02 현재 용접시간 / R02 표준시간 최소 용접시간 설정
LOAD      F0009A
AND>      D018010 D008321	// R02 현재 용접시간 / R02 표준시간 최대 용접시간
OR LOAD
AND LOAD
AND<=     D008323 D008322	// R02 W10 RH 용접구간 카운터설정 / R02 W10 RH 용접구간 카운터
AND NOT   D015012.2	// R02 Weld Count By_Pass On
MOVP      2 D006010	// R02 W10 RH 용접누락 판정결과
MLOAD
AND>=     D018010 D008320	// R02 현재 용접시간 / R02 표준시간 최소 용접시간 설정
LOAD<=    D018010 D008321	// R02 현재 용접시간 / R02 표준시간 최대 용접시간
OR        F00099
AND LOAD
AND>      D008323 D008322	// R02 W10 RH 용접구간 카운터설정 / R02 W10 RH 용접구간 카운터
AND NOT   D015012.2	// R02 Weld Count By_Pass On
MOVP      3 D006010	// R02 W10 RH 용접누락 판정결과
MPOP
LOAD<     D018010 D008320	// R02 현재 용접시간 / R02 표준시간 최소 용접시간 설정
LOAD      F0009A
AND>      D018010 D008321	// R02 현재 용접시간 / R02 표준시간 최대 용접시간
OR LOAD
AND LOAD
AND>      D008323 D008322	// R02 W10 RH 용접구간 카운터설정 / R02 W10 RH 용접구간 카운터
AND NOT   D015012.2	// R02 Weld Count By_Pass On
MOVP      4 D006010	// R02 W10 RH 용접누락 판정결과
; L416
LOAD NOT  P10209	// R02 Arc_On -> PLC
MOV       0 D018018	// R02 용접누락 진행상태
; L417
LOAD NOT  P10210	// R02 (OT01) W10 RH 간섭무
AND       P10209	// R02 Arc_On -> PLC
MOV       1 D018018	// R02 용접누락 진행상태

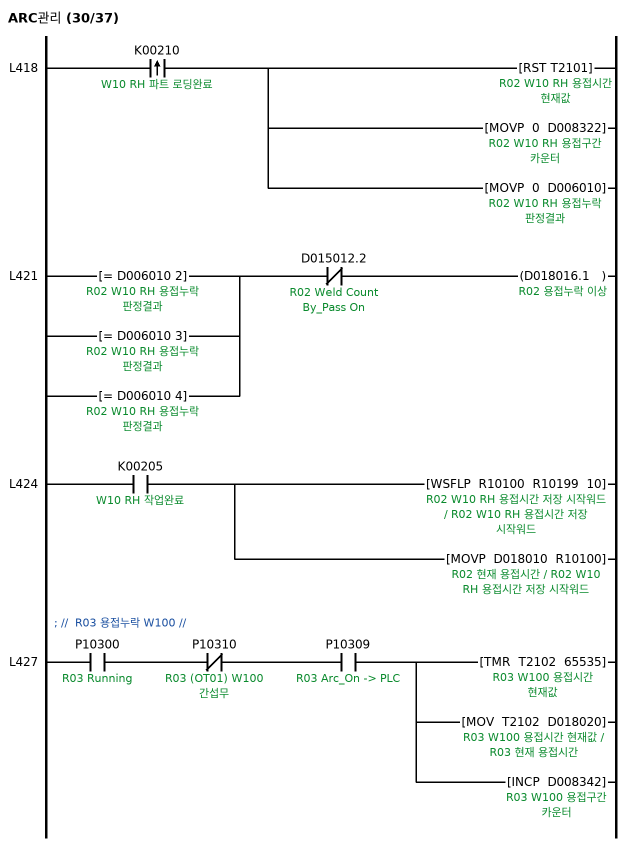
; L418
LOADP     K00210	// W10 RH 파트 로딩완료
RST       T2101	// R02 W10 RH 용접시간 현재값
MOVP      0 D008322	// R02 W10 RH 용접구간 카운터
MOVP      0 D006010	// R02 W10 RH 용접누락 판정결과
; L421
LOAD=     D006010 2	// R02 W10 RH 용접누락 판정결과
OR=       D006010 3	// R02 W10 RH 용접누락 판정결과
OR=       D006010 4	// R02 W10 RH 용접누락 판정결과
AND NOT   D015012.2	// R02 Weld Count By_Pass On
OUT       D018016.1	// R02 용접누락 이상
; L424
LOAD      K00205	// W10 RH 작업완료
WSFLP     R10100 R10199 10	// R02 W10 RH 용접시간 저장 시작워드 / R02 W10 RH 용접시간 저장 시작워드
MOVP      D018010 R10100	// R02 현재 용접시간 / R02 W10 RH 용접시간 저장 시작워드
//   //  R03 용접누락 W100 //
; L427
LOAD      P10300	// R03 Running
AND NOT   P10310	// R03 (OT01) W100 간섭무
AND       P10309	// R03 Arc_On -> PLC
TMR       T2102 65535	// R03 W100 용접시간 현재값
MOV       T2102 D018020	// R03 W100 용접시간 현재값 / R03 현재 용접시간
INCP      D008342	// R03 W100 용접구간 카운터

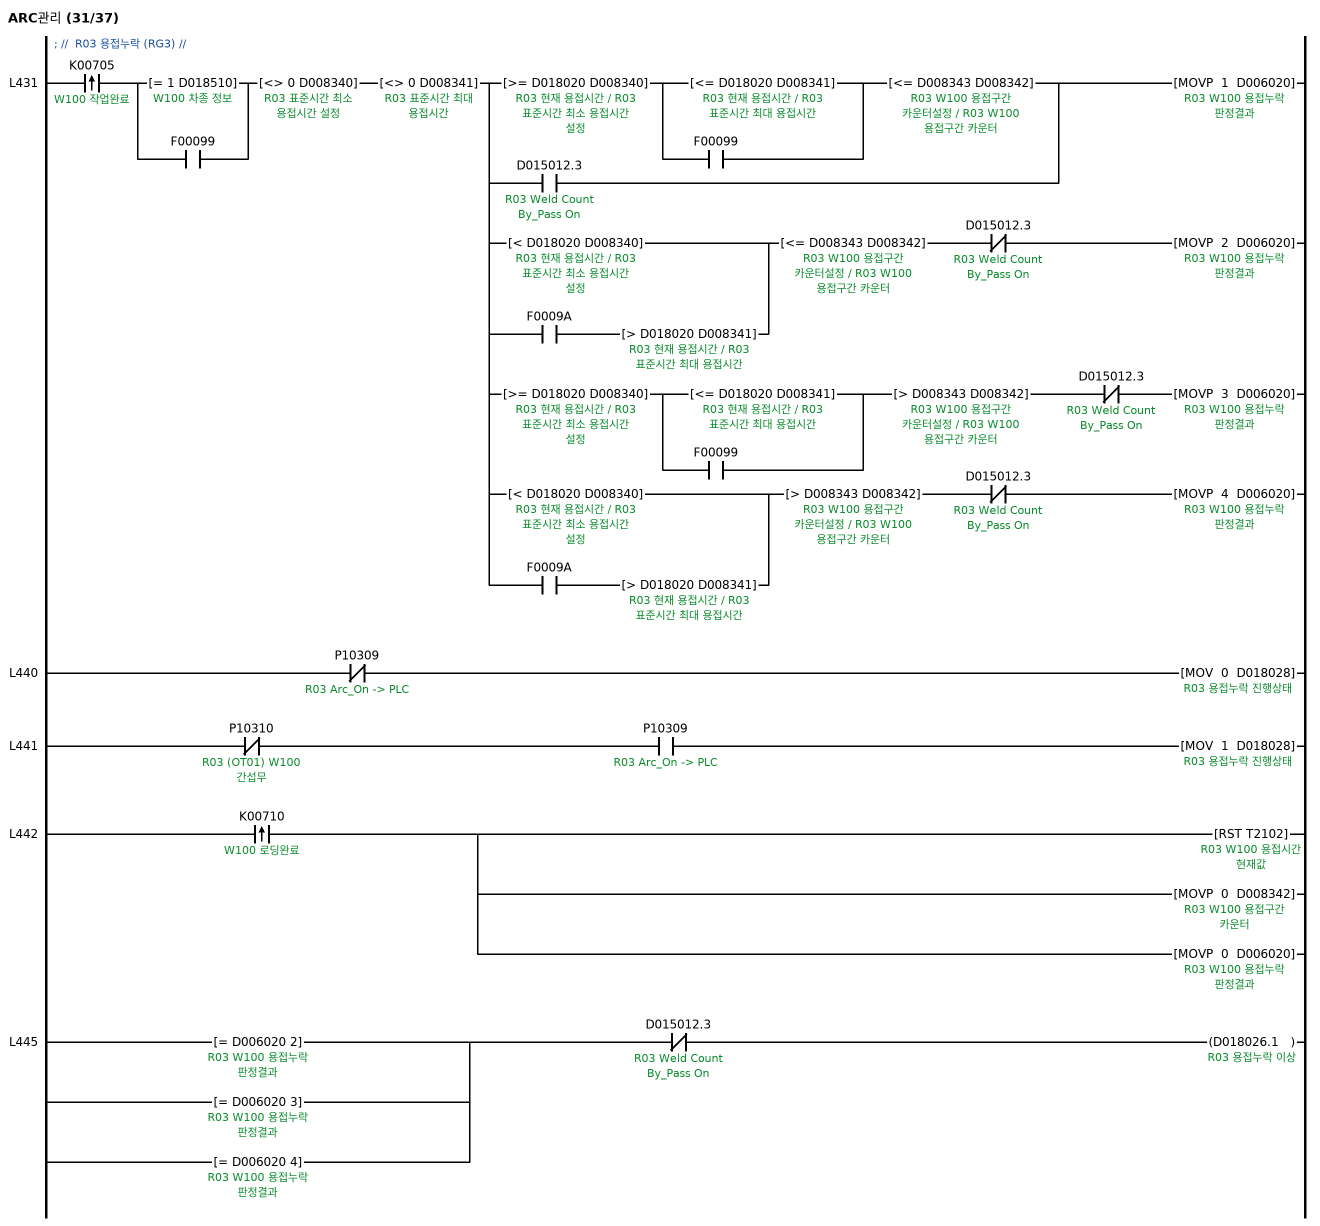
//   //  R03 용접누락 (RG3) //
; L431
LOADP     K00705	// W100 작업완료
LOAD=     1 D018510	// W100 차종 정보
OR        F00099
AND LOAD
AND<>     0 D008340	// R03 표준시간 최소 용접시간 설정
AND<>     0 D008341	// R03 표준시간 최대 용접시간
MPUSH
LOAD>=    D018020 D008340	// R03 현재 용접시간 / R03 표준시간 최소 용접시간 설정
LOAD<=    D018020 D008341	// R03 현재 용접시간 / R03 표준시간 최대 용접시간
OR        F00099
AND LOAD
AND<=     D008343 D008342	// R03 W100 용접구간 카운터설정 / R03 W100 용접구간 카운터
OR        D015012.3	// R03 Weld Count By_Pass On
AND LOAD
MOVP      1 D006020	// R03 W100 용접누락 판정결과
MLOAD
LOAD<     D018020 D008340	// R03 현재 용접시간 / R03 표준시간 최소 용접시간 설정
LOAD      F0009A
AND>      D018020 D008341	// R03 현재 용접시간 / R03 표준시간 최대 용접시간
OR LOAD
AND LOAD
AND<=     D008343 D008342	// R03 W100 용접구간 카운터설정 / R03 W100 용접구간 카운터
AND NOT   D015012.3	// R03 Weld Count By_Pass On
MOVP      2 D006020	// R03 W100 용접누락 판정결과
MLOAD
AND>=     D018020 D008340	// R03 현재 용접시간 / R03 표준시간 최소 용접시간 설정
LOAD<=    D018020 D008341	// R03 현재 용접시간 / R03 표준시간 최대 용접시간
OR        F00099
AND LOAD
AND>      D008343 D008342	// R03 W100 용접구간 카운터설정 / R03 W100 용접구간 카운터
AND NOT   D015012.3	// R03 Weld Count By_Pass On
MOVP      3 D006020	// R03 W100 용접누락 판정결과
MPOP
LOAD<     D018020 D008340	// R03 현재 용접시간 / R03 표준시간 최소 용접시간 설정
LOAD      F0009A
AND>      D018020 D008341	// R03 현재 용접시간 / R03 표준시간 최대 용접시간
OR LOAD
AND LOAD
AND>      D008343 D008342	// R03 W100 용접구간 카운터설정 / R03 W100 용접구간 카운터
AND NOT   D015012.3	// R03 Weld Count By_Pass On
MOVP      4 D006020	// R03 W100 용접누락 판정결과
; L440
LOAD NOT  P10309	// R03 Arc_On -> PLC
MOV       0 D018028	// R03 용접누락 진행상태
; L441
LOAD NOT  P10310	// R03 (OT01) W100 간섭무
AND       P10309	// R03 Arc_On -> PLC
MOV       1 D018028	// R03 용접누락 진행상태
; L442
LOADP     K00710	// W100 로딩완료
RST       T2102	// R03 W100 용접시간 현재값
MOVP      0 D008342	// R03 W100 용접구간 카운터
MOVP      0 D006020	// R03 W100 용접누락 판정결과
; L445
LOAD=     D006020 2	// R03 W100 용접누락 판정결과
OR=       D006020 3	// R03 W100 용접누락 판정결과
OR=       D006020 4	// R03 W100 용접누락 판정결과
AND NOT   D015012.3	// R03 Weld Count By_Pass On
OUT       D018026.1	// R03 용접누락 이상

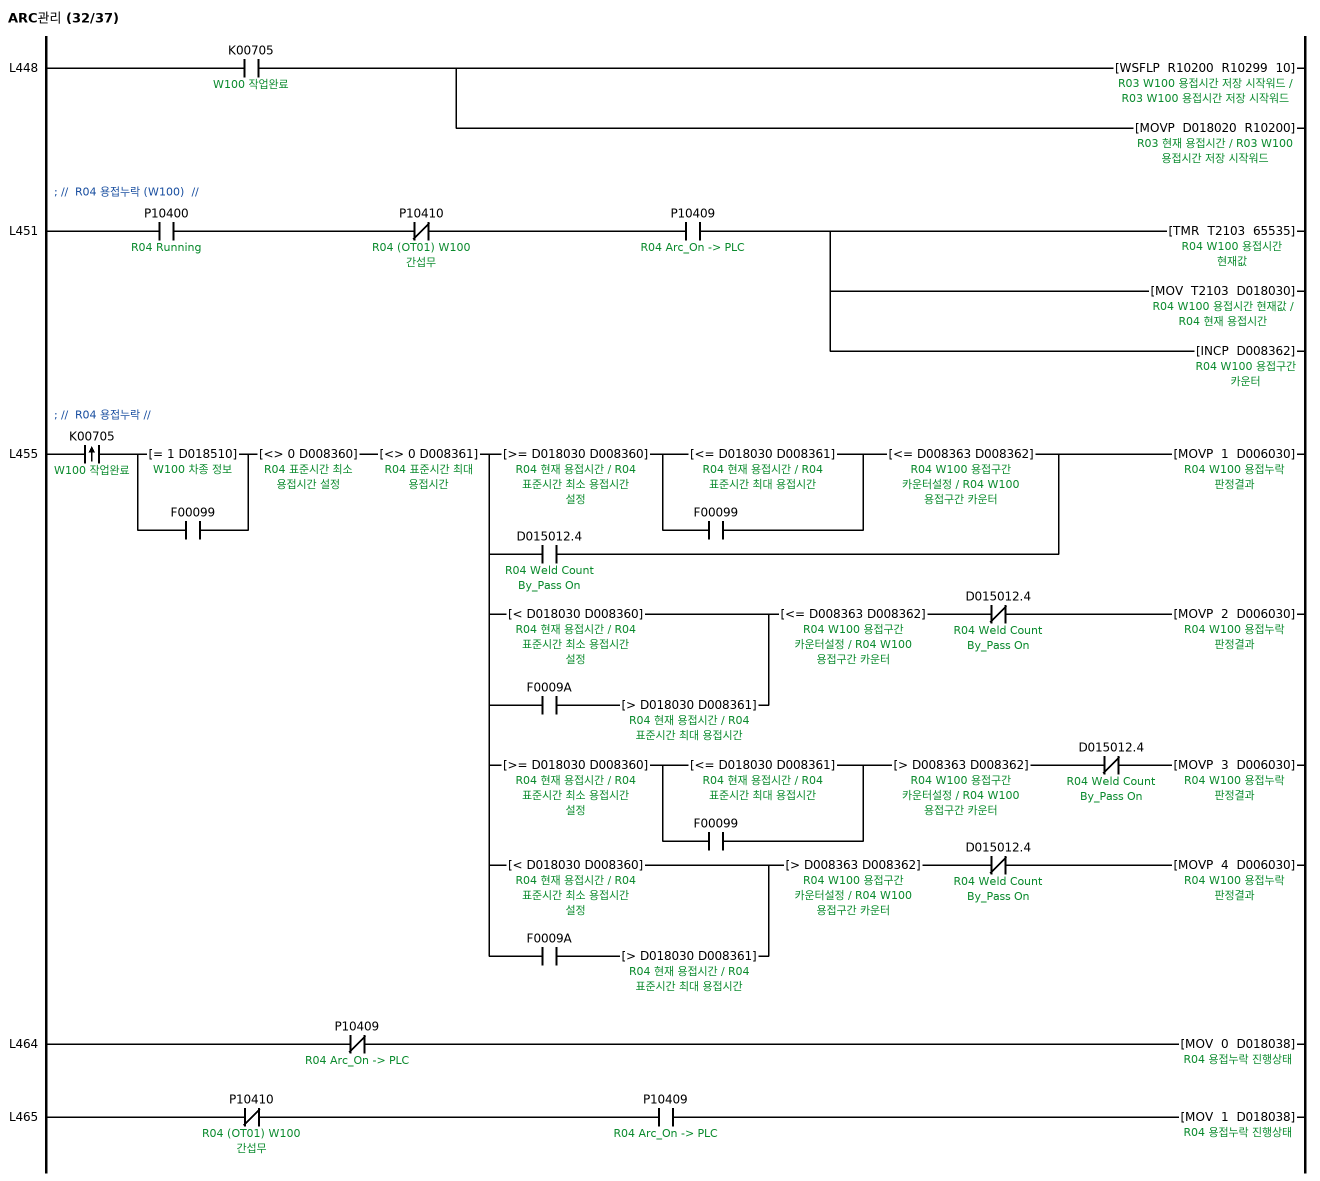
; L448
LOAD      K00705	// W100 작업완료
WSFLP     R10200 R10299 10	// R03 W100 용접시간 저장 시작워드 / R03 W100 용접시간 저장 시작워드
MOVP      D018020 R10200	// R03 현재 용접시간 / R03 W100 용접시간 저장 시작워드
//   //  R04 용접누락 (W100)  //
; L451
LOAD      P10400	// R04 Running
AND NOT   P10410	// R04 (OT01) W100 간섭무
AND       P10409	// R04 Arc_On -> PLC
TMR       T2103 65535	// R04 W100 용접시간 현재값
MOV       T2103 D018030	// R04 W100 용접시간 현재값 / R04 현재 용접시간
INCP      D008362	// R04 W100 용접구간 카운터
//   //  R04 용접누락 //
; L455
LOADP     K00705	// W100 작업완료
LOAD=     1 D018510	// W100 차종 정보
OR        F00099
AND LOAD
AND<>     0 D008360	// R04 표준시간 최소 용접시간 설정
AND<>     0 D008361	// R04 표준시간 최대 용접시간
MPUSH
LOAD>=    D018030 D008360	// R04 현재 용접시간 / R04 표준시간 최소 용접시간 설정
LOAD<=    D018030 D008361	// R04 현재 용접시간 / R04 표준시간 최대 용접시간
OR        F00099
AND LOAD
AND<=     D008363 D008362	// R04 W100 용접구간 카운터설정 / R04 W100 용접구간 카운터
OR        D015012.4	// R04 Weld Count By_Pass On
AND LOAD
MOVP      1 D006030	// R04 W100 용접누락 판정결과
MLOAD
LOAD<     D018030 D008360	// R04 현재 용접시간 / R04 표준시간 최소 용접시간 설정
LOAD      F0009A
AND>      D018030 D008361	// R04 현재 용접시간 / R04 표준시간 최대 용접시간
OR LOAD
AND LOAD
AND<=     D008363 D008362	// R04 W100 용접구간 카운터설정 / R04 W100 용접구간 카운터
AND NOT   D015012.4	// R04 Weld Count By_Pass On
MOVP      2 D006030	// R04 W100 용접누락 판정결과
MLOAD
AND>=     D018030 D008360	// R04 현재 용접시간 / R04 표준시간 최소 용접시간 설정
LOAD<=    D018030 D008361	// R04 현재 용접시간 / R04 표준시간 최대 용접시간
OR        F00099
AND LOAD
AND>      D008363 D008362	// R04 W100 용접구간 카운터설정 / R04 W100 용접구간 카운터
AND NOT   D015012.4	// R04 Weld Count By_Pass On
MOVP      3 D006030	// R04 W100 용접누락 판정결과
MPOP
LOAD<     D018030 D008360	// R04 현재 용접시간 / R04 표준시간 최소 용접시간 설정
LOAD      F0009A
AND>      D018030 D008361	// R04 현재 용접시간 / R04 표준시간 최대 용접시간
OR LOAD
AND LOAD
AND>      D008363 D008362	// R04 W100 용접구간 카운터설정 / R04 W100 용접구간 카운터
AND NOT   D015012.4	// R04 Weld Count By_Pass On
MOVP      4 D006030	// R04 W100 용접누락 판정결과
; L464
LOAD NOT  P10409	// R04 Arc_On -> PLC
MOV       0 D018038	// R04 용접누락 진행상태
; L465
LOAD NOT  P10410	// R04 (OT01) W100 간섭무
AND       P10409	// R04 Arc_On -> PLC
MOV       1 D018038	// R04 용접누락 진행상태

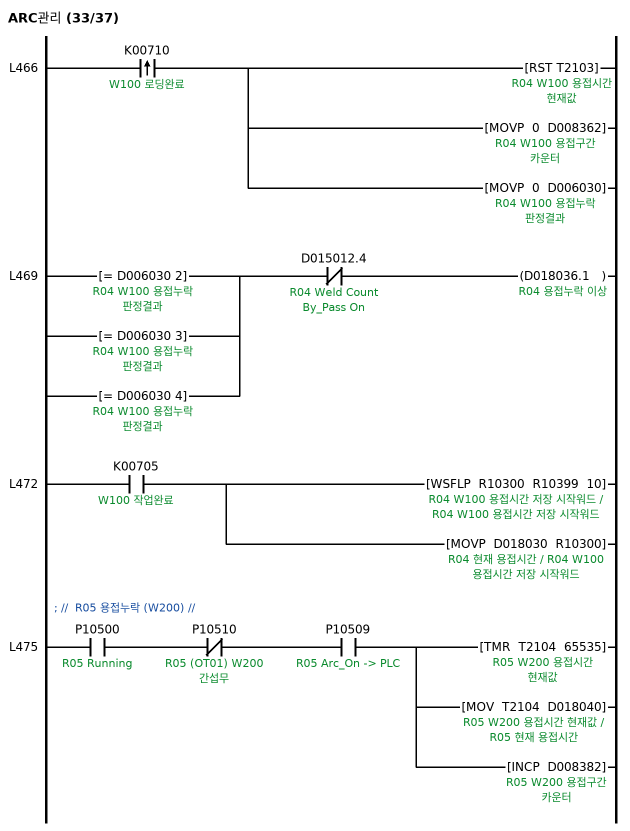
; L466
LOADP     K00710	// W100 로딩완료
RST       T2103	// R04 W100 용접시간 현재값
MOVP      0 D008362	// R04 W100 용접구간 카운터
MOVP      0 D006030	// R04 W100 용접누락 판정결과
; L469
LOAD=     D006030 2	// R04 W100 용접누락 판정결과
OR=       D006030 3	// R04 W100 용접누락 판정결과
OR=       D006030 4	// R04 W100 용접누락 판정결과
AND NOT   D015012.4	// R04 Weld Count By_Pass On
OUT       D018036.1	// R04 용접누락 이상
; L472
LOAD      K00705	// W100 작업완료
WSFLP     R10300 R10399 10	// R04 W100 용접시간 저장 시작워드 / R04 W100 용접시간 저장 시작워드
MOVP      D018030 R10300	// R04 현재 용접시간 / R04 W100 용접시간 저장 시작워드
//   //  R05 용접누락 (W200) //
; L475
LOAD      P10500	// R05 Running
AND NOT   P10510	// R05 (OT01) W200 간섭무
AND       P10509	// R05 Arc_On -> PLC
TMR       T2104 65535	// R05 W200 용접시간 현재값
MOV       T2104 D018040	// R05 W200 용접시간 현재값 / R05 현재 용접시간
INCP      D008382	// R05 W200 용접구간 카운터

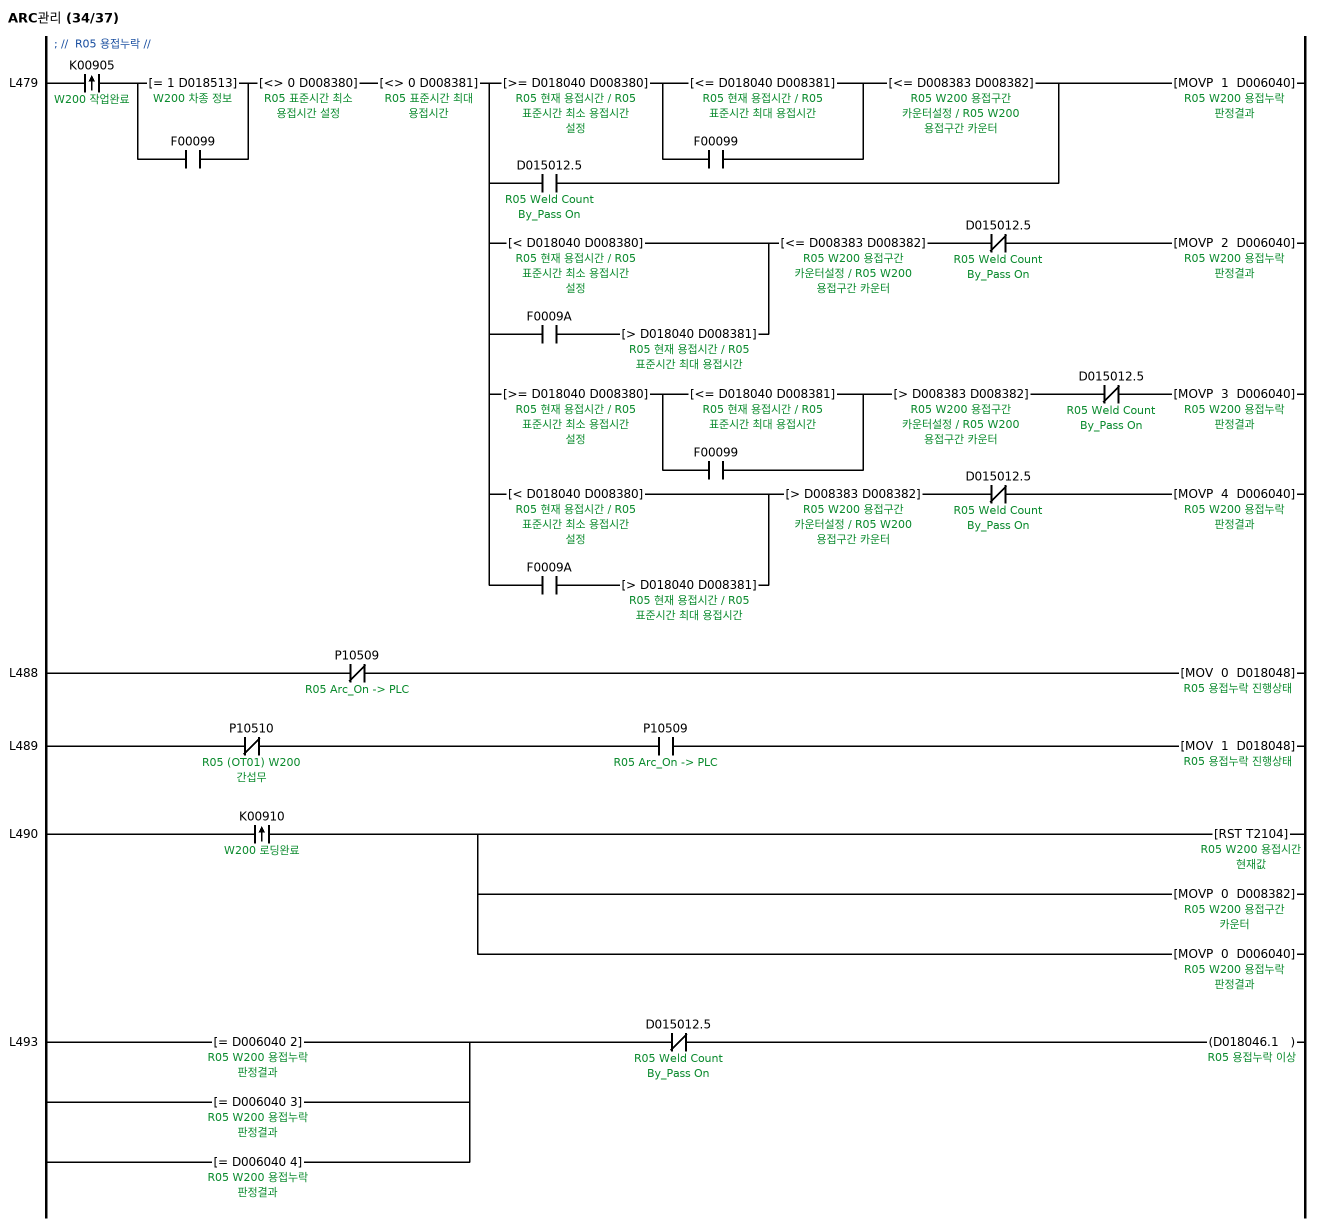
//   //  R05 용접누락 //
; L479
LOADP     K00905	// W200 작업완료
LOAD=     1 D018513	// W200 차종 정보
OR        F00099
AND LOAD
AND<>     0 D008380	// R05 표준시간 최소 용접시간 설정
AND<>     0 D008381	// R05 표준시간 최대 용접시간
MPUSH
LOAD>=    D018040 D008380	// R05 현재 용접시간 / R05 표준시간 최소 용접시간 설정
LOAD<=    D018040 D008381	// R05 현재 용접시간 / R05 표준시간 최대 용접시간
OR        F00099
AND LOAD
AND<=     D008383 D008382	// R05 W200 용접구간 카운터설정 / R05 W200 용접구간 카운터
OR        D015012.5	// R05 Weld Count By_Pass On
AND LOAD
MOVP      1 D006040	// R05 W200 용접누락 판정결과
MLOAD
LOAD<     D018040 D008380	// R05 현재 용접시간 / R05 표준시간 최소 용접시간 설정
LOAD      F0009A
AND>      D018040 D008381	// R05 현재 용접시간 / R05 표준시간 최대 용접시간
OR LOAD
AND LOAD
AND<=     D008383 D008382	// R05 W200 용접구간 카운터설정 / R05 W200 용접구간 카운터
AND NOT   D015012.5	// R05 Weld Count By_Pass On
MOVP      2 D006040	// R05 W200 용접누락 판정결과
MLOAD
AND>=     D018040 D008380	// R05 현재 용접시간 / R05 표준시간 최소 용접시간 설정
LOAD<=    D018040 D008381	// R05 현재 용접시간 / R05 표준시간 최대 용접시간
OR        F00099
AND LOAD
AND>      D008383 D008382	// R05 W200 용접구간 카운터설정 / R05 W200 용접구간 카운터
AND NOT   D015012.5	// R05 Weld Count By_Pass On
MOVP      3 D006040	// R05 W200 용접누락 판정결과
MPOP
LOAD<     D018040 D008380	// R05 현재 용접시간 / R05 표준시간 최소 용접시간 설정
LOAD      F0009A
AND>      D018040 D008381	// R05 현재 용접시간 / R05 표준시간 최대 용접시간
OR LOAD
AND LOAD
AND>      D008383 D008382	// R05 W200 용접구간 카운터설정 / R05 W200 용접구간 카운터
AND NOT   D015012.5	// R05 Weld Count By_Pass On
MOVP      4 D006040	// R05 W200 용접누락 판정결과
; L488
LOAD NOT  P10509	// R05 Arc_On -> PLC
MOV       0 D018048	// R05 용접누락 진행상태
; L489
LOAD NOT  P10510	// R05 (OT01) W200 간섭무
AND       P10509	// R05 Arc_On -> PLC
MOV       1 D018048	// R05 용접누락 진행상태
; L490
LOADP     K00910	// W200 로딩완료
RST       T2104	// R05 W200 용접시간 현재값
MOVP      0 D008382	// R05 W200 용접구간 카운터
MOVP      0 D006040	// R05 W200 용접누락 판정결과
; L493
LOAD=     D006040 2	// R05 W200 용접누락 판정결과
OR=       D006040 3	// R05 W200 용접누락 판정결과
OR=       D006040 4	// R05 W200 용접누락 판정결과
AND NOT   D015012.5	// R05 Weld Count By_Pass On
OUT       D018046.1	// R05 용접누락 이상

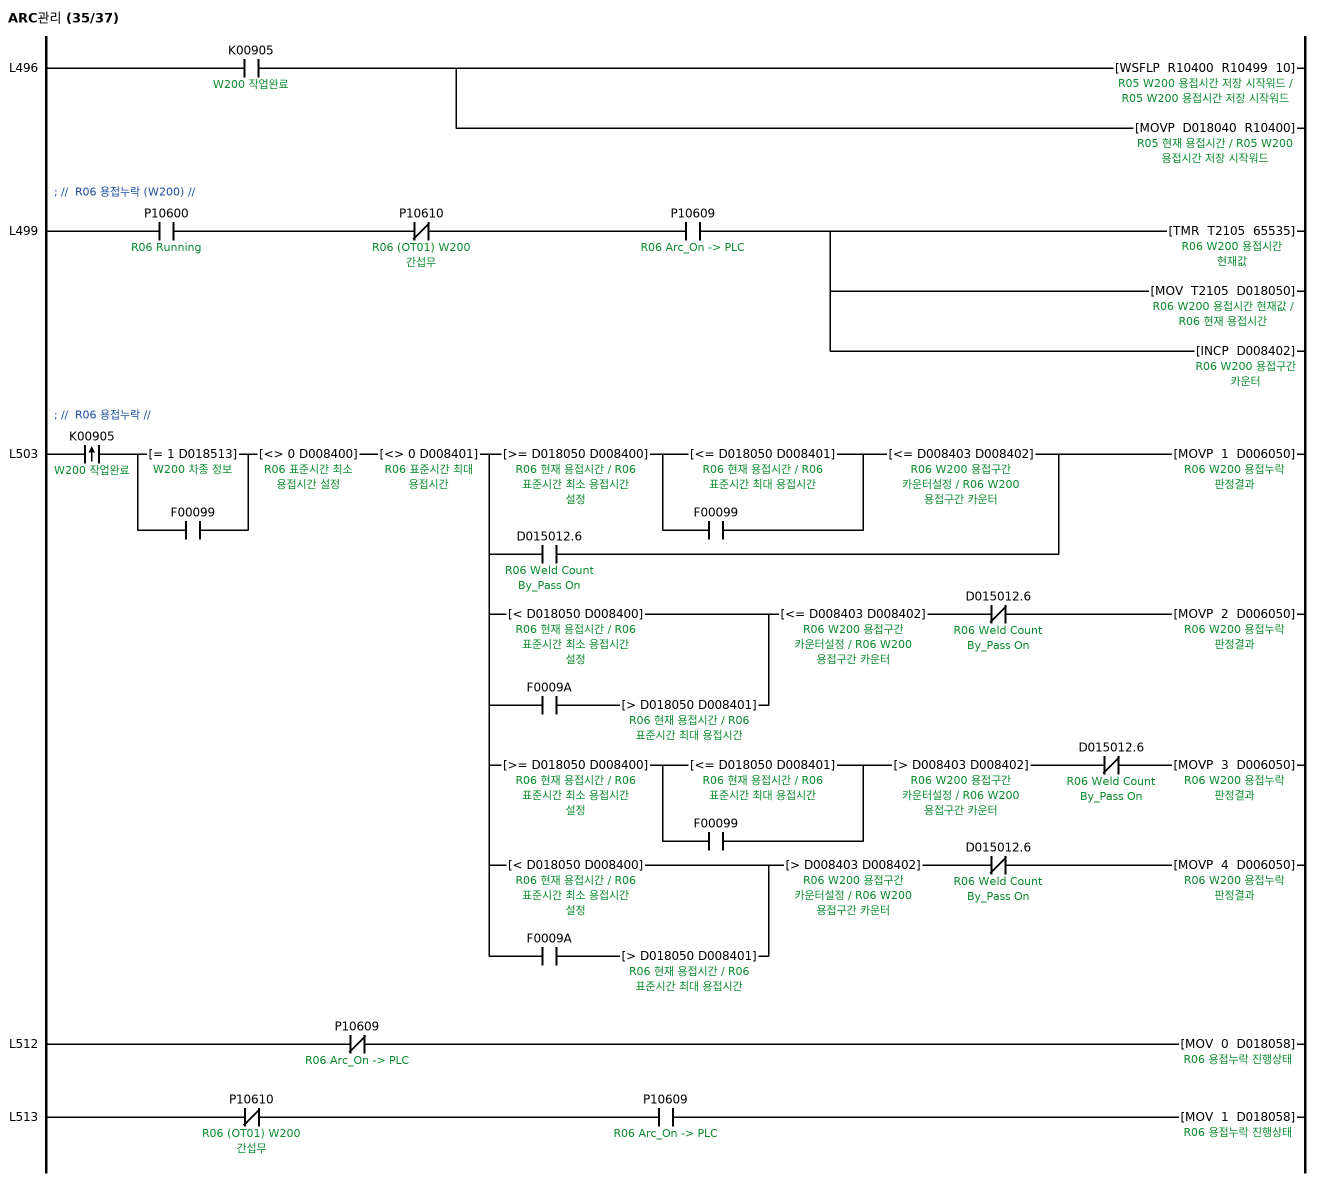
; L496
LOAD      K00905	// W200 작업완료
WSFLP     R10400 R10499 10	// R05 W200 용접시간 저장 시작워드 / R05 W200 용접시간 저장 시작워드
MOVP      D018040 R10400	// R05 현재 용접시간 / R05 W200 용접시간 저장 시작워드
//   //  R06 용접누락 (W200) //
; L499
LOAD      P10600	// R06 Running
AND NOT   P10610	// R06 (OT01) W200 간섭무
AND       P10609	// R06 Arc_On -> PLC
TMR       T2105 65535	// R06 W200 용접시간 현재값
MOV       T2105 D018050	// R06 W200 용접시간 현재값 / R06 현재 용접시간
INCP      D008402	// R06 W200 용접구간 카운터
//   //  R06 용접누락 //
; L503
LOADP     K00905	// W200 작업완료
LOAD=     1 D018513	// W200 차종 정보
OR        F00099
AND LOAD
AND<>     0 D008400	// R06 표준시간 최소 용접시간 설정
AND<>     0 D008401	// R06 표준시간 최대 용접시간
MPUSH
LOAD>=    D018050 D008400	// R06 현재 용접시간 / R06 표준시간 최소 용접시간 설정
LOAD<=    D018050 D008401	// R06 현재 용접시간 / R06 표준시간 최대 용접시간
OR        F00099
AND LOAD
AND<=     D008403 D008402	// R06 W200 용접구간 카운터설정 / R06 W200 용접구간 카운터
OR        D015012.6	// R06 Weld Count By_Pass On
AND LOAD
MOVP      1 D006050	// R06 W200 용접누락 판정결과
MLOAD
LOAD<     D018050 D008400	// R06 현재 용접시간 / R06 표준시간 최소 용접시간 설정
LOAD      F0009A
AND>      D018050 D008401	// R06 현재 용접시간 / R06 표준시간 최대 용접시간
OR LOAD
AND LOAD
AND<=     D008403 D008402	// R06 W200 용접구간 카운터설정 / R06 W200 용접구간 카운터
AND NOT   D015012.6	// R06 Weld Count By_Pass On
MOVP      2 D006050	// R06 W200 용접누락 판정결과
MLOAD
AND>=     D018050 D008400	// R06 현재 용접시간 / R06 표준시간 최소 용접시간 설정
LOAD<=    D018050 D008401	// R06 현재 용접시간 / R06 표준시간 최대 용접시간
OR        F00099
AND LOAD
AND>      D008403 D008402	// R06 W200 용접구간 카운터설정 / R06 W200 용접구간 카운터
AND NOT   D015012.6	// R06 Weld Count By_Pass On
MOVP      3 D006050	// R06 W200 용접누락 판정결과
MPOP
LOAD<     D018050 D008400	// R06 현재 용접시간 / R06 표준시간 최소 용접시간 설정
LOAD      F0009A
AND>      D018050 D008401	// R06 현재 용접시간 / R06 표준시간 최대 용접시간
OR LOAD
AND LOAD
AND>      D008403 D008402	// R06 W200 용접구간 카운터설정 / R06 W200 용접구간 카운터
AND NOT   D015012.6	// R06 Weld Count By_Pass On
MOVP      4 D006050	// R06 W200 용접누락 판정결과
; L512
LOAD NOT  P10609	// R06 Arc_On -> PLC
MOV       0 D018058	// R06 용접누락 진행상태
; L513
LOAD NOT  P10610	// R06 (OT01) W200 간섭무
AND       P10609	// R06 Arc_On -> PLC
MOV       1 D018058	// R06 용접누락 진행상태

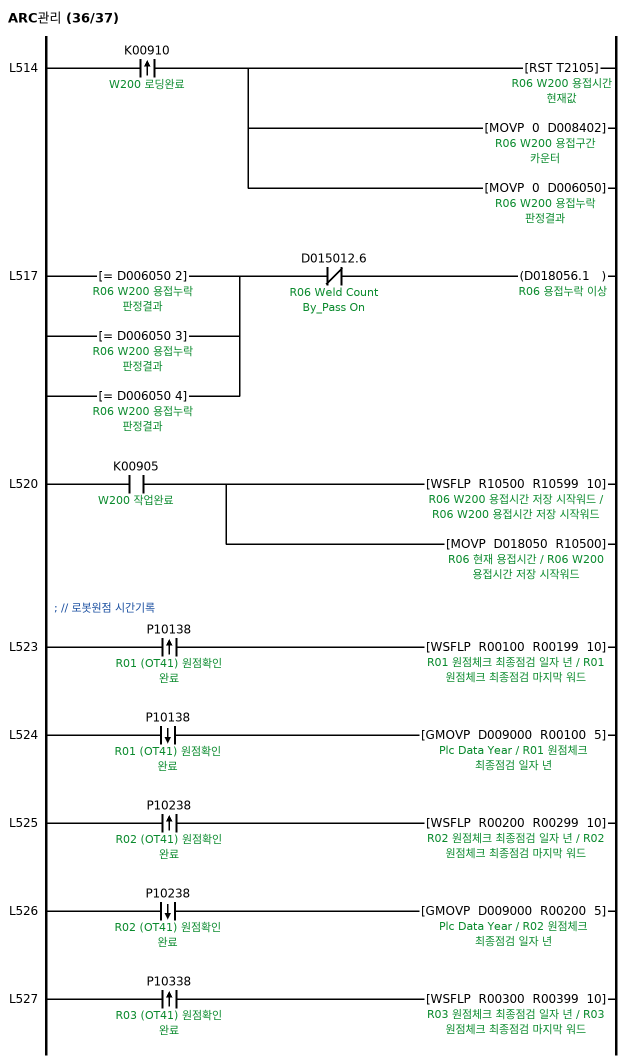
; L514
LOADP     K00910	// W200 로딩완료
RST       T2105	// R06 W200 용접시간 현재값
MOVP      0 D008402	// R06 W200 용접구간 카운터
MOVP      0 D006050	// R06 W200 용접누락 판정결과
; L517
LOAD=     D006050 2	// R06 W200 용접누락 판정결과
OR=       D006050 3	// R06 W200 용접누락 판정결과
OR=       D006050 4	// R06 W200 용접누락 판정결과
AND NOT   D015012.6	// R06 Weld Count By_Pass On
OUT       D018056.1	// R06 용접누락 이상
; L520
LOAD      K00905	// W200 작업완료
WSFLP     R10500 R10599 10	// R06 W200 용접시간 저장 시작워드 / R06 W200 용접시간 저장 시작워드
MOVP      D018050 R10500	// R06 현재 용접시간 / R06 W200 용접시간 저장 시작워드
// // 로봇원점 시간기록
; L523
LOADP     P10138	// R01 (OT41) 원점확인 완료
WSFLP     R00100 R00199 10	// R01 원점체크 최종점검 일자 년 / R01 원점체크 최종점검 마지막 워드
; L524
LOADN     P10138	// R01 (OT41) 원점확인 완료
GMOVP     D009000 R00100 5	// Plc Data Year / R01 원점체크 최종점검 일자 년
; L525
LOADP     P10238	// R02 (OT41) 원점확인 완료
WSFLP     R00200 R00299 10	// R02 원점체크 최종점검 일자 년 / R02 원점체크 최종점검 마지막 워드
; L526
LOADN     P10238	// R02 (OT41) 원점확인 완료
GMOVP     D009000 R00200 5	// Plc Data Year / R02 원점체크 최종점검 일자 년
; L527
LOADP     P10338	// R03 (OT41) 원점확인 완료
WSFLP     R00300 R00399 10	// R03 원점체크 최종점검 일자 년 / R03 원점체크 최종점검 마지막 워드

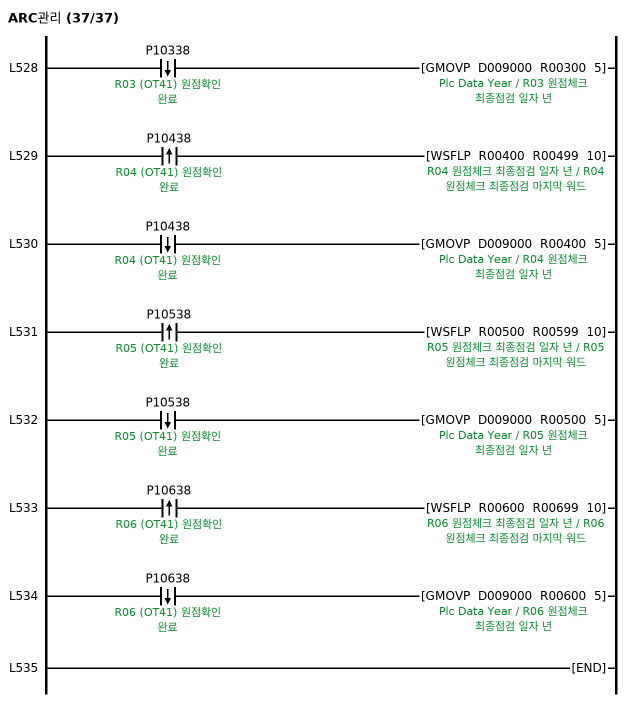
; L528
LOADN     P10338	// R03 (OT41) 원점확인 완료
GMOVP     D009000 R00300 5	// Plc Data Year / R03 원점체크 최종점검 일자 년
; L529
LOADP     P10438	// R04 (OT41) 원점확인 완료
WSFLP     R00400 R00499 10	// R04 원점체크 최종점검 일자 년 / R04 원점체크 최종점검 마지막 워드
; L530
LOADN     P10438	// R04 (OT41) 원점확인 완료
GMOVP     D009000 R00400 5	// Plc Data Year / R04 원점체크 최종점검 일자 년
; L531
LOADP     P10538	// R05 (OT41) 원점확인 완료
WSFLP     R00500 R00599 10	// R05 원점체크 최종점검 일자 년 / R05 원점체크 최종점검 마지막 워드
; L532
LOADN     P10538	// R05 (OT41) 원점확인 완료
GMOVP     D009000 R00500 5	// Plc Data Year / R05 원점체크 최종점검 일자 년
; L533
LOADP     P10638	// R06 (OT41) 원점확인 완료
WSFLP     R00600 R00699 10	// R06 원점체크 최종점검 일자 년 / R06 원점체크 최종점검 마지막 워드
; L534
LOADN     P10638	// R06 (OT41) 원점확인 완료
GMOVP     D009000 R00600 5	// Plc Data Year / R06 원점체크 최종점검 일자 년
; L535
END

PROGRAM 차종데이타_트래킹 (task: 스캔 프로그램)

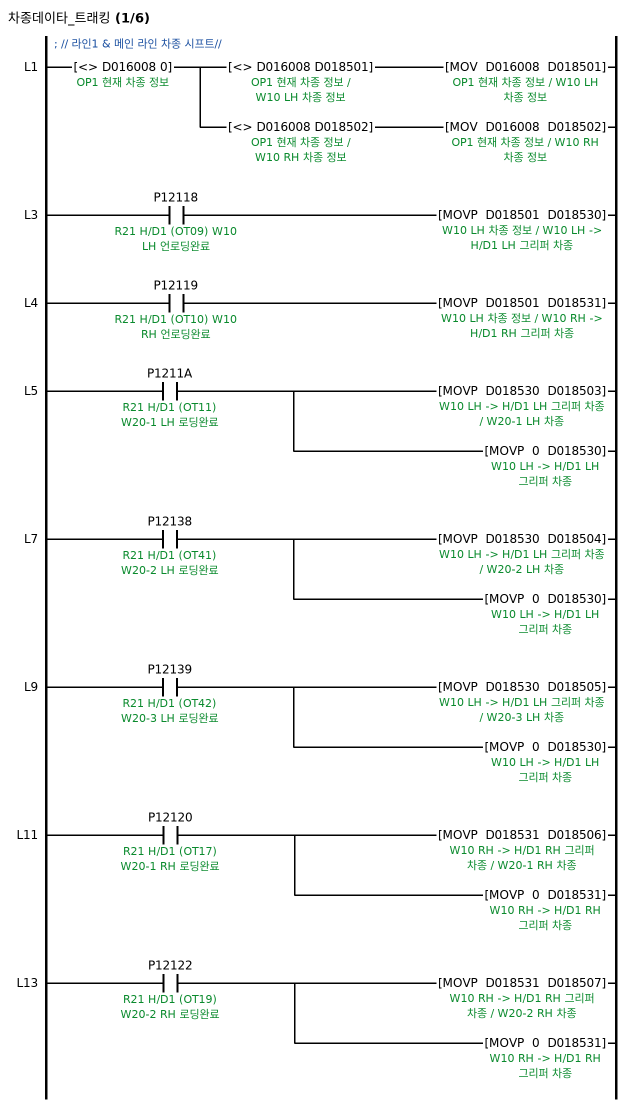
// // 라인1 & 메인 라인 차종 시프트//
; L1
LOAD<>    D016008 0	// OP1 현재 차종 정보
MPUSH
AND<>     D016008 D018501	// OP1 현재 차종 정보 / W10 LH 차종 정보
MOV       D016008 D018501	// OP1 현재 차종 정보 / W10 LH 차종 정보
MPOP
AND<>     D016008 D018502	// OP1 현재 차종 정보 / W10 RH 차종 정보
MOV       D016008 D018502	// OP1 현재 차종 정보 / W10 RH 차종 정보
; L3
LOAD      P12118	// R21 H/D1 (OT09) W10 LH 언로딩완료
MOVP      D018501 D018530	// W10 LH 차종 정보 / W10 LH -> H/D1 LH 그리퍼 차종
; L4
LOAD      P12119	// R21 H/D1 (OT10) W10 RH 언로딩완료
MOVP      D018501 D018531	// W10 LH 차종 정보 / W10 RH -> H/D1 RH 그리퍼 차종
; L5
LOAD      P1211A	// R21 H/D1 (OT11) W20-1 LH 로딩완료
MOVP      D018530 D018503	// W10 LH -> H/D1 LH 그리퍼 차종 / W20-1 LH 차종
MOVP      0 D018530	// W10 LH -> H/D1 LH 그리퍼 차종
; L7
LOAD      P12138	// R21 H/D1 (OT41) W20-2 LH 로딩완료
MOVP      D018530 D018504	// W10 LH -> H/D1 LH 그리퍼 차종 / W20-2 LH 차종
MOVP      0 D018530	// W10 LH -> H/D1 LH 그리퍼 차종
; L9
LOAD      P12139	// R21 H/D1 (OT42) W20-3 LH 로딩완료
MOVP      D018530 D018505	// W10 LH -> H/D1 LH 그리퍼 차종 / W20-3 LH 차종
MOVP      0 D018530	// W10 LH -> H/D1 LH 그리퍼 차종
; L11
LOAD      P12120	// R21 H/D1 (OT17) W20-1 RH 로딩완료
MOVP      D018531 D018506	// W10 RH -> H/D1 RH 그리퍼 차종 / W20-1 RH 차종
MOVP      0 D018531	// W10 RH -> H/D1 RH 그리퍼 차종
; L13
LOAD      P12122	// R21 H/D1 (OT19) W20-2 RH 로딩완료
MOVP      D018531 D018507	// W10 RH -> H/D1 RH 그리퍼 차종 / W20-2 RH 차종
MOVP      0 D018531	// W10 RH -> H/D1 RH 그리퍼 차종

